LIN {X -288.759,Y -26.804,Z 58.424,A 5.303,B 90.000,C 0.000} C_DIS
LIN {X -288.763,Y -26.761,Z 58.730,A 5.295,B 90.000,C 0.000} C_DIS
LIN {X -288.767,Y -26.710,Z 58.794,A 5.285,B 90.000,C 0.000} C_DIS
LIN {X -288.772,Y -26.660,Z 58.836,A 5.275,B 90.000,C 0.000} C_DIS
LIN {X -288.776,Y -26.617,Z 59.040,A 5.266,B 90.000,C 0.000} C_DIS
LIN {X -288.781,Y -26.567,Z 59.083,A 5.256,B 90.000,C 0.000} C_DIS
LIN {X -288.785,Y -26.516,Z 59.147,A 5.246,B 90.000,C 0.000} C_DIS
LIN {X -288.789,Y -26.473,Z 59.453,A 5.238,B 90.000,C 0.000} C_DIS
LIN {X -288.794,Y -26.423,Z 59.516,A 5.228,B 90.000,C 0.000} C_DIS
LIN {X -288.798,Y -26.372,Z 59.559,A 5.218,B 90.000,C 0.000} C_DIS
LIN {X -288.802,Y -26.330,Z 59.763,A 5.209,B 90.000,C 0.000} C_DIS
LIN {X -288.807,Y -26.279,Z 59.805,A 5.199,B 90.000,C 0.000} C_DIS
LIN {X -288.812,Y -26.228,Z 59.869,A 5.189,B 90.000,C 0.000} C_DIS
LIN {X -288.815,Y -26.186,Z 60.175,A 5.181,B 90.000,C 0.000} C_DIS
LIN {X -288.825,Y -26.084,Z 60.303,A 5.160,B 90.000,C 0.000} C_DIS
LIN {X -288.828,Y -26.042,Z 60.609,A 5.152,B 90.000,C 0.000} C_DIS
LIN {X -288.833,Y -25.991,Z 60.673,A 5.142,B 90.000,C 0.000} C_DIS
LIN {X -288.838,Y -25.940,Z 60.715,A 5.132,B 90.000,C 0.000} C_DIS
LIN {X -288.841,Y -25.898,Z 60.919,A 5.123,B 90.000,C 0.000} C_DIS
LIN {X -288.846,Y -25.847,Z 60.962,A 5.113,B 90.000,C 0.000} C_DIS
LIN {X -288.850,Y -25.796,Z 61.025,A 5.103,B 90.000,C 0.000} C_DIS
LIN {X -288.854,Y -25.754,Z 61.332,A 5.095,B 90.000,C 0.000} C_DIS
LIN {X -288.859,Y -25.703,Z 61.395,A 5.085,B 90.000,C 0.000} C_DIS
LIN {X -288.863,Y -25.652,Z 61.438,A 5.075,B 90.000,C 0.000} C_DIS
LIN {X -288.867,Y -25.610,Z 61.642,A 5.066,B 90.000,C 0.000} C_DIS
LIN {X -288.871,Y -25.559,Z 61.684,A 5.056,B 90.000,C 0.000} C_DIS
LIN {X -288.876,Y -25.508,Z 61.748,A 5.046,B 90.000,C 0.000} C_DIS
LIN {X -288.880,Y -25.466,Z 62.054,A 5.038,B 90.000,C 0.000} C_DIS
LIN {X -288.884,Y -25.415,Z 62.118,A 5.028,B 90.000,C 0.000} C_DIS
LIN {X -288.889,Y -25.364,Z 62.160,A 5.018,B 90.000,C 0.000} C_DIS
LIN {X -288.892,Y -25.322,Z 62.365,A 5.009,B 90.000,C 0.000} C_DIS
LIN {X -288.897,Y -25.271,Z 62.407,A 4.999,B 90.000,C 0.000} C_DIS
LIN {X -288.901,Y -25.220,Z 62.471,A 4.989,B 90.000,C 0.000} C_DIS
LIN {X -288.905,Y -25.178,Z 62.777,A 4.981,B 90.000,C 0.000} C_DIS
LIN {X -288.909,Y -25.127,Z 62.841,A 4.971,B 90.000,C 0.000} C_DIS
LIN {X -288.914,Y -25.076,Z 62.883,A 4.961,B 90.000,C 0.000} C_DIS
LIN {X -288.917,Y -25.034,Z 63.087,A 4.952,B 90.000,C 0.000} C_DIS
LIN {X -288.922,Y -24.983,Z 63.130,A 4.942,B 90.000,C 0.000} C_DIS
LIN {X -288.926,Y -24.932,Z 63.193,A 4.932,B 90.000,C 0.000} C_DIS
LIN {X -288.930,Y -24.890,Z 63.500,A 4.924,B 90.000,C 0.000} C_DIS
LIN {X -288.934,Y -24.839,Z 63.563,A 4.914,B 90.000,C 0.000} C_DIS
LIN {X -288.939,Y -24.788,Z 63.606,A 4.903,B 90.000,C 0.000} C_DIS
LIN {X -288.942,Y -24.746,Z 63.810,A 4.895,B 90.000,C 0.000} C_DIS
LIN {X -288.947,Y -24.695,Z 63.852,A 4.885,B 90.000,C 0.000} C_DIS
LIN {X -288.951,Y -24.644,Z 63.916,A 4.875,B 90.000,C 0.000} C_DIS
LIN {X -288.955,Y -24.602,Z 64.222,A 4.866,B 90.000,C 0.000} C_DIS
LIN {X -288.959,Y -24.551,Z 64.286,A 4.856,B 90.000,C 0.000} C_DIS
LIN {X -288.963,Y -24.500,Z 64.328,A 4.846,B 90.000,C 0.000} C_DIS
LIN {X -288.967,Y -24.458,Z 64.532,A 4.838,B 90.000,C 0.000} C_DIS
LIN {X -288.971,Y -24.407,Z 64.575,A 4.828,B 90.000,C 0.000} C_DIS
LIN {X -288.975,Y -24.356,Z 64.639,A 4.818,B 90.000,C 0.000} C_DIS
LIN {X -288.979,Y -24.314,Z 64.945,A 4.809,B 90.000,C 0.000} C_DIS
LIN {X -288.983,Y -24.263,Z 65.009,A 4.799,B 90.000,C 0.000} C_DIS
LIN {X -288.987,Y -24.212,Z 65.051,A 4.789,B 90.000,C 0.000} C_DIS
LIN {X -288.991,Y -24.170,Z 65.255,A 4.781,B 90.000,C 0.000} C_DIS
LIN {X -288.995,Y -24.119,Z 65.298,A 4.771,B 90.000,C 0.000} C_DIS
LIN {X -289.000,Y -24.068,Z 65.361,A 4.761,B 90.000,C 0.000} C_DIS
LIN {X -289.003,Y -24.026,Z 65.667,A 4.752,B 90.000,C 0.000} C_DIS
LIN {X -289.007,Y -23.975,Z 65.731,A 4.742,B 90.000,C 0.000} C_DIS
LIN {X -289.011,Y -23.924,Z 65.774,A 4.732,B 90.000,C 0.000} C_DIS
LIN {X -289.015,Y -23.882,Z 65.978,A 4.724,B 90.000,C 0.000} C_DIS
LIN {X -289.019,Y -23.831,Z 66.020,A 4.714,B 90.000,C 0.000} C_DIS
LIN {X -289.023,Y -23.780,Z 66.084,A 4.704,B 90.000,C 0.000} C_DIS
LIN {X -289.027,Y -23.738,Z 66.390,A 4.695,B 90.000,C 0.000} C_DIS
LIN {X -289.031,Y -23.687,Z 66.454,A 4.685,B 90.000,C 0.000} C_DIS
LIN {X -289.035,Y -23.636,Z 66.496,A 4.675,B 90.000,C 0.000} C_DIS
LIN {X -289.039,Y -23.594,Z 66.700,A 4.667,B 90.000,C 0.000} C_DIS
LIN {X -289.043,Y -23.543,Z 66.743,A 4.657,B 90.000,C 0.000} C_DIS
LIN {X -289.047,Y -23.492,Z 66.807,A 4.646,B 90.000,C 0.000} C_DIS
LIN {X -289.050,Y -23.450,Z 67.113,A 4.638,B 90.000,C 0.000} C_DIS
LIN {X -289.054,Y -23.399,Z 67.176,A 4.628,B 90.000,C 0.000} C_DIS
LIN {X -289.059,Y -23.348,Z 67.219,A 4.618,B 90.000,C 0.000} C_DIS
LIN {X -289.062,Y -23.306,Z 67.423,A 4.609,B 90.000,C 0.000} C_DIS
LIN {X -289.066,Y -23.255,Z 67.465,A 4.599,B 90.000,C 0.000} C_DIS
LIN {X -289.070,Y -23.204,Z 67.529,A 4.589,B 90.000,C 0.000} C_DIS
LIN {X -289.074,Y -23.162,Z 67.835,A 4.581,B 90.000,C 0.000} C_DIS
LIN {X -289.078,Y -23.111,Z 67.899,A 4.571,B 90.000,C 0.000} C_DIS
LIN {X -289.082,Y -23.060,Z 67.942,A 4.561,B 90.000,C 0.000} C_DIS
LIN {X -289.085,Y -23.017,Z 68.146,A 4.552,B 90.000,C 0.000} C_DIS
LIN {X -289.089,Y -22.967,Z 68.188,A 4.542,B 90.000,C 0.000} C_DIS
LIN {X -289.093,Y -22.916,Z 68.252,A 4.532,B 90.000,C 0.000} C_DIS
LIN {X -289.097,Y -22.873,Z 68.558,A 4.524,B 90.000,C 0.000} C_DIS
LIN {X -289.101,Y -22.822,Z 68.622,A 4.514,B 90.000,C 0.000} C_DIS
LIN {X -289.105,Y -22.772,Z 68.664,A 4.504,B 90.000,C 0.000} C_DIS
LIN {X -289.108,Y -22.729,Z 68.868,A 4.495,B 90.000,C 0.000} C_DIS
LIN {X -289.112,Y -22.678,Z 68.911,A 4.485,B 90.000,C 0.000} C_DIS
LIN {X -289.116,Y -22.628,Z 68.974,A 4.475,B 90.000,C 0.000} C_DIS
LIN {X -289.119,Y -22.585,Z 69.281,A 4.467,B 90.000,C 0.000} C_DIS
LIN {X -289.123,Y -22.534,Z 69.344,A 4.457,B 90.000,C 0.000} C_DIS
LIN {X -289.127,Y -22.483,Z 69.387,A 4.447,B 90.000,C 0.000} C_DIS
LIN {X -289.130,Y -22.441,Z 69.591,A 4.438,B 90.000,C 0.000} C_DIS
LIN {X -289.134,Y -22.390,Z 69.633,A 4.428,B 90.000,C 0.000} C_DIS
LIN {X -289.138,Y -22.339,Z 69.697,A 4.418,B 90.000,C 0.000} C_DIS
LIN {X -289.142,Y -22.297,Z 70.003,A 4.410,B 90.000,C 0.000} C_DIS
LIN {X -289.145,Y -22.246,Z 70.067,A 4.400,B 90.000,C 0.000} C_DIS
LIN {X -289.149,Y -22.195,Z 70.109,A 4.389,B 90.000,C 0.000} C_DIS
LIN {X -289.153,Y -22.153,Z 70.314,A 4.381,B 90.000,C 0.000} C_DIS
LIN {X -289.157,Y -22.102,Z 70.356,A 4.371,B 90.000,C 0.000} C_DIS
LIN {X -289.160,Y -22.051,Z 70.420,A 4.361,B 90.000,C 0.000} C_DIS
LIN {X -289.164,Y -22.009,Z 70.726,A 4.353,B 90.000,C 0.000} C_DIS
LIN {X -289.168,Y -21.958,Z 70.790,A 4.342,B 90.000,C 0.000} C_DIS
LIN {X -289.171,Y -21.907,Z 70.832,A 4.332,B 90.000,C 0.000} C_DIS
LIN {X -289.175,Y -21.865,Z 71.036,A 4.324,B 90.000,C 0.000} C_DIS
LIN {X -289.178,Y -21.814,Z 71.079,A 4.314,B 90.000,C 0.000} C_DIS
LIN {X -289.182,Y -21.763,Z 71.142,A 4.304,B 90.000,C 0.000} C_DIS
LIN {X -289.185,Y -21.721,Z 71.449,A 4.295,B 90.000,C 0.000} C_DIS
LIN {X -289.189,Y -21.670,Z 71.512,A 4.285,B 90.000,C 0.000} C_DIS
LIN {X -289.193,Y -21.619,Z 71.555,A 4.275,B 90.000,C 0.000} C_DIS
LIN {X -289.196,Y -21.576,Z 71.759,A 4.267,B 90.000,C 0.000} C_DIS
LIN {X -289.200,Y -21.526,Z 71.801,A 4.257,B 90.000,C 0.000} C_DIS
LIN {X -289.204,Y -21.475,Z 71.865,A 4.247,B 90.000,C 0.000} C_DIS
LIN {X -289.207,Y -21.432,Z 72.171,A 4.238,B 90.000,C 0.000} C_DIS
LIN {X -289.211,Y -21.381,Z 72.235,A 4.228,B 90.000,C 0.000} C_DIS
LIN {X -289.214,Y -21.331,Z 72.277,A 4.218,B 90.000,C 0.000} C_DIS
LIN {X -289.218,Y -21.288,Z 72.482,A 4.210,B 90.000,C 0.000} C_DIS
LIN {X -289.221,Y -21.237,Z 72.524,A 4.200,B 90.000,C 0.000} C_DIS
LIN {X -289.225,Y -21.186,Z 72.588,A 4.190,B 90.000,C 0.000} C_DIS
LIN {X -289.228,Y -21.144,Z 72.894,A 4.181,B 90.000,C 0.000} C_DIS
LIN {X -289.236,Y -21.042,Z 73.021,A 4.161,B 90.000,C 0.000} C_DIS
LIN {X -289.239,Y -21.000,Z 73.327,A 4.153,B 90.000,C 0.000} C_DIS
LIN {X -289.242,Y -20.949,Z 73.391,A 4.143,B 90.000,C 0.000} C_DIS
LIN {X -289.246,Y -20.898,Z 73.434,A 4.132,B 90.000,C 0.000} C_DIS
LIN {X -289.249,Y -20.856,Z 73.638,A 4.124,B 90.000,C 0.000} C_DIS
LIN {X -289.253,Y -20.805,Z 73.680,A 4.114,B 90.000,C 0.000} C_DIS
LIN {X -289.256,Y -20.754,Z 73.744,A 4.104,B 90.000,C 0.000} C_DIS
LIN {X -289.259,Y -20.712,Z 74.050,A 4.096,B 90.000,C 0.000} C_DIS
LIN {X -289.263,Y -20.661,Z 74.114,A 4.085,B 90.000,C 0.000} C_DIS
LIN {X -289.267,Y -20.610,Z 74.156,A 4.075,B 90.000,C 0.000} C_DIS
LIN {X -289.270,Y -20.567,Z 74.360,A 4.067,B 90.000,C 0.000} C_DIS
LIN {X -289.273,Y -20.517,Z 74.403,A 4.057,B 90.000,C 0.000} C_DIS
LIN {X -289.277,Y -20.466,Z 74.467,A 4.047,B 90.000,C 0.000} C_DIS
LIN {X -289.280,Y -20.423,Z 74.773,A 4.038,B 90.000,C 0.000} C_DIS
LIN {X -289.284,Y -20.372,Z 74.836,A 4.028,B 90.000,C 0.000} C_DIS
LIN {X -289.287,Y -20.321,Z 74.879,A 4.018,B 90.000,C 0.000} C_DIS
LIN {X -289.290,Y -20.279,Z 75.083,A 4.010,B 90.000,C 0.000} C_DIS
LIN {X -289.294,Y -20.228,Z 75.125,A 4.000,B 90.000,C 0.000} C_DIS
LIN {X -289.297,Y -20.177,Z 75.189,A 3.990,B 90.000,C 0.000} C_DIS
LIN {X -289.300,Y -20.135,Z 75.495,A 3.981,B 90.000,C 0.000} C_DIS
LIN {X -289.304,Y -20.084,Z 75.559,A 3.971,B 90.000,C 0.000} C_DIS
LIN {X -289.307,Y -20.033,Z 75.602,A 3.961,B 90.000,C 0.000} C_DIS
LIN {X -289.310,Y -19.991,Z 75.806,A 3.953,B 90.000,C 0.000} C_DIS
LIN {X -289.314,Y -19.940,Z 75.848,A 3.943,B 90.000,C 0.000} C_DIS
LIN {X -289.317,Y -19.889,Z 75.912,A 3.933,B 90.000,C 0.000} C_DIS
LIN {X -289.320,Y -19.847,Z 76.218,A 3.924,B 90.000,C 0.000} C_DIS
LIN {X -289.324,Y -19.796,Z 76.282,A 3.914,B 90.000,C 0.000} C_DIS
LIN {X -289.327,Y -19.745,Z 76.324,A 3.904,B 90.000,C 0.000} C_DIS
LIN {X -289.330,Y -19.702,Z 76.528,A 3.896,B 90.000,C 0.000} C_DIS
LIN {X -289.333,Y -19.651,Z 76.571,A 3.886,B 90.000,C 0.000} C_DIS
LIN {X -289.337,Y -19.601,Z 76.634,A 3.875,B 90.000,C 0.000} C_DIS
LIN {X -289.340,Y -19.558,Z 76.941,A 3.867,B 90.000,C 0.000} C_DIS
LIN {X -289.343,Y -19.507,Z 77.004,A 3.857,B 90.000,C 0.000} C_DIS
LIN {X -289.347,Y -19.456,Z 77.047,A 3.847,B 90.000,C 0.000} C_DIS
LIN {X -289.349,Y -19.414,Z 77.251,A 3.839,B 90.000,C 0.000} C_DIS
LIN {X -289.353,Y -19.363,Z 77.293,A 3.828,B 90.000,C 0.000} C_DIS
LIN {X -289.356,Y -19.312,Z 77.357,A 3.818,B 90.000,C 0.000} C_DIS
LIN {X -289.359,Y -19.270,Z 77.663,A 3.810,B 90.000,C 0.000} C_DIS
LIN {X -289.362,Y -19.219,Z 77.727,A 3.800,B 90.000,C 0.000} C_DIS
LIN {X -289.366,Y -19.168,Z 77.769,A 3.790,B 90.000,C 0.000} C_DIS
LIN {X -289.369,Y -19.126,Z 77.974,A 3.781,B 90.000,C 0.000} C_DIS
LIN {X -289.372,Y -19.075,Z 78.016,A 3.771,B 90.000,C 0.000} C_DIS
LIN {X -289.375,Y -19.024,Z 78.080,A 3.761,B 90.000,C 0.000} C_DIS
LIN {X -289.378,Y -18.981,Z 78.386,A 3.753,B 90.000,C 0.000} C_DIS
LIN {X -289.381,Y -18.930,Z 78.450,A 3.743,B 90.000,C 0.000} C_DIS
LIN {X -289.385,Y -18.879,Z 78.492,A 3.733,B 90.000,C 0.000} C_DIS
LIN {X -289.388,Y -18.837,Z 78.696,A 3.724,B 90.000,C 0.000} C_DIS
LIN {X -289.391,Y -18.786,Z 78.739,A 3.714,B 90.000,C 0.000} C_DIS
LIN {X -289.394,Y -18.735,Z 78.802,A 3.704,B 90.000,C 0.000} C_DIS
LIN {X -289.397,Y -18.693,Z 79.109,A 3.696,B 90.000,C 0.000} C_DIS
LIN {X -289.400,Y -18.642,Z 79.172,A 3.686,B 90.000,C 0.000} C_DIS
LIN {X -289.403,Y -18.591,Z 79.215,A 3.676,B 90.000,C 0.000} C_DIS
LIN {X -289.406,Y -18.549,Z 79.419,A 3.667,B 90.000,C 0.000} C_DIS
LIN {X -289.409,Y -18.498,Z 79.461,A 3.657,B 90.000,C 0.000} C_DIS
LIN {X -289.413,Y -18.447,Z 79.525,A 3.647,B 90.000,C 0.000} C_DIS
LIN {X -289.415,Y -18.404,Z 79.831,A 3.639,B 90.000,C 0.000} C_DIS
LIN {X -289.419,Y -18.353,Z 79.895,A 3.629,B 90.000,C 0.000} C_DIS
LIN {X -289.422,Y -18.303,Z 79.937,A 3.618,B 90.000,C 0.000} C_DIS
LIN {X -289.425,Y -18.260,Z 80.142,A 3.610,B 90.000,C 0.000} C_DIS
LIN {X -289.428,Y -18.209,Z 80.184,A 3.600,B 90.000,C 0.000} C_DIS
LIN {X -289.431,Y -18.158,Z 80.248,A 3.590,B 90.000,C 0.000} C_DIS
LIN {X -289.434,Y -18.116,Z 80.554,A 3.582,B 90.000,C 0.000} C_DIS
LIN {X -289.437,Y -18.065,Z 80.618,A 3.571,B 90.000,C 0.000} C_DIS
LIN {X -289.440,Y -18.014,Z 80.660,A 3.561,B 90.000,C 0.000} C_DIS
LIN {X -289.443,Y -17.972,Z 80.864,A 3.553,B 90.000,C 0.000} C_DIS
LIN {X -289.446,Y -17.921,Z 80.907,A 3.543,B 90.000,C 0.000} C_DIS
LIN {X -289.449,Y -17.870,Z 80.970,A 3.533,B 90.000,C 0.000} C_DIS
LIN {X -289.452,Y -17.827,Z 81.277,A 3.524,B 90.000,C 0.000} C_DIS
LIN {X -289.455,Y -17.776,Z 81.340,A 3.514,B 90.000,C 0.000} C_DIS
LIN {X -289.458,Y -17.726,Z 81.383,A 3.504,B 90.000,C 0.000} C_DIS
LIN {X -289.460,Y -17.683,Z 81.587,A 3.496,B 90.000,C 0.000} C_DIS
LIN {X -289.463,Y -17.632,Z 81.629,A 3.486,B 90.000,C 0.000} C_DIS
LIN {X -289.467,Y -17.581,Z 81.693,A 3.476,B 90.000,C 0.000} C_DIS
LIN {X -289.469,Y -17.539,Z 81.999,A 3.467,B 90.000,C 0.000} C_DIS
LIN {X -289.472,Y -17.488,Z 82.063,A 3.457,B 90.000,C 0.000} C_DIS
LIN {X -289.475,Y -17.437,Z 82.105,A 3.447,B 90.000,C 0.000} C_DIS
LIN {X -289.478,Y -17.395,Z 82.309,A 3.439,B 90.000,C 0.000} C_DIS
LIN {X -289.481,Y -17.344,Z 82.352,A 3.429,B 90.000,C 0.000} C_DIS
LIN {X -289.484,Y -17.293,Z 82.416,A 3.419,B 90.000,C 0.000} C_DIS
LIN {X -289.486,Y -17.250,Z 82.722,A 3.410,B 90.000,C 0.000} C_DIS
LIN {X -289.490,Y -17.199,Z 82.785,A 3.400,B 90.000,C 0.000} C_DIS
LIN {X -289.493,Y -17.148,Z 82.828,A 3.390,B 90.000,C 0.000} C_DIS
LIN {X -289.495,Y -17.106,Z 83.032,A 3.382,B 90.000,C 0.000} C_DIS
LIN {X -289.498,Y -17.055,Z 83.075,A 3.372,B 90.000,C 0.000} C_DIS
LIN {X -289.501,Y -17.004,Z 83.138,A 3.361,B 90.000,C 0.000} C_DIS
LIN {X -289.504,Y -16.962,Z 83.444,A 3.353,B 90.000,C 0.000} C_DIS
LIN {X -289.507,Y -16.911,Z 83.508,A 3.343,B 90.000,C 0.000} C_DIS
LIN {X -289.509,Y -16.860,Z 83.551,A 3.333,B 90.000,C 0.000} C_DIS
LIN {X -289.512,Y -16.818,Z 83.755,A 3.325,B 90.000,C 0.000} C_DIS
LIN {X -289.515,Y -16.767,Z 83.797,A 3.314,B 90.000,C 0.000} C_DIS
LIN {X -289.518,Y -16.716,Z 83.861,A 3.304,B 90.000,C 0.000} C_DIS
LIN {X -289.520,Y -16.673,Z 84.167,A 3.296,B 90.000,C 0.000} C_DIS
LIN {X -289.523,Y -16.622,Z 84.231,A 3.286,B 90.000,C 0.000} C_DIS
LIN {X -289.526,Y -16.571,Z 84.273,A 3.276,B 90.000,C 0.000} C_DIS
LIN {X -289.529,Y -16.529,Z 84.477,A 3.267,B 90.000,C 0.000} C_DIS
LIN {X -289.531,Y -16.478,Z 84.520,A 3.257,B 90.000,C 0.000} C_DIS
LIN {X -289.534,Y -16.427,Z 84.584,A 3.247,B 90.000,C 0.000} C_DIS
LIN {X -289.537,Y -16.385,Z 84.890,A 3.239,B 90.000,C 0.000} C_DIS
LIN {X -289.543,Y -16.283,Z 85.017,A 3.219,B 90.000,C 0.000} C_DIS
LIN {X -289.545,Y -16.240,Z 85.323,A 3.210,B 90.000,C 0.000} C_DIS
LIN {X -289.548,Y -16.189,Z 85.387,A 3.200,B 90.000,C 0.000} C_DIS
LIN {X -289.551,Y -16.138,Z 85.429,A 3.190,B 90.000,C 0.000} C_DIS
LIN {X -289.553,Y -16.096,Z 85.634,A 3.182,B 90.000,C 0.000} C_DIS
LIN {X -289.556,Y -16.045,Z 85.676,A 3.172,B 90.000,C 0.000} C_DIS
LIN {X -289.559,Y -15.994,Z 85.740,A 3.162,B 90.000,C 0.000} C_DIS
LIN {X -289.561,Y -15.952,Z 86.046,A 3.153,B 90.000,C 0.000} C_DIS
LIN {X -289.564,Y -15.901,Z 86.110,A 3.143,B 90.000,C 0.000} C_DIS
LIN {X -289.567,Y -15.850,Z 86.152,A 3.133,B 90.000,C 0.000} C_DIS
LIN {X -289.569,Y -15.807,Z 86.356,A 3.125,B 90.000,C 0.000} C_DIS
LIN {X -289.572,Y -15.756,Z 86.399,A 3.115,B 90.000,C 0.000} C_DIS
LIN {X -289.574,Y -15.706,Z 86.462,A 3.104,B 90.000,C 0.000} C_DIS
LIN {X -289.577,Y -15.663,Z 86.769,A 3.096,B 90.000,C 0.000} C_DIS
LIN {X -289.579,Y -15.612,Z 86.832,A 3.086,B 90.000,C 0.000} C_DIS
LIN {X -289.582,Y -15.561,Z 86.875,A 3.076,B 90.000,C 0.000} C_DIS
LIN {X -289.584,Y -15.519,Z 87.079,A 3.068,B 90.000,C 0.000} C_DIS
LIN {X -289.587,Y -15.468,Z 87.121,A 3.057,B 90.000,C 0.000} C_DIS
LIN {X -289.590,Y -15.417,Z 87.185,A 3.047,B 90.000,C 0.000} C_DIS
LIN {X -289.592,Y -15.374,Z 87.491,A 3.039,B 90.000,C 0.000} C_DIS
LIN {X -289.595,Y -15.324,Z 87.555,A 3.029,B 90.000,C 0.000} C_DIS
LIN {X -289.598,Y -15.273,Z 87.597,A 3.019,B 90.000,C 0.000} C_DIS
LIN {X -289.600,Y -15.230,Z 87.802,A 3.010,B 90.000,C 0.000} C_DIS
LIN {X -289.602,Y -15.179,Z 87.844,A 3.000,B 90.000,C 0.000} C_DIS
LIN {X -289.605,Y -15.128,Z 87.908,A 2.990,B 90.000,C 0.000} C_DIS
LIN {X -289.607,Y -15.086,Z 88.214,A 2.982,B 90.000,C 0.000} C_DIS
LIN {X -289.610,Y -15.035,Z 88.278,A 2.972,B 90.000,C 0.000} C_DIS
LIN {X -289.613,Y -14.984,Z 88.320,A 2.962,B 90.000,C 0.000} C_DIS
LIN {X -289.615,Y -14.941,Z 88.524,A 2.953,B 90.000,C 0.000} C_DIS
LIN {X -289.617,Y -14.891,Z 88.567,A 2.943,B 90.000,C 0.000} C_DIS
LIN {X -289.620,Y -14.840,Z 88.630,A 2.933,B 90.000,C 0.000} C_DIS
LIN {X -289.622,Y -14.797,Z 88.937,A 2.925,B 90.000,C 0.000} C_DIS
LIN {X -289.625,Y -14.746,Z 89.000,A 2.915,B 90.000,C 0.000} C_DIS
LIN {X -289.627,Y -14.695,Z 89.043,A 2.905,B 90.000,C 0.000} C_DIS
LIN {X -289.630,Y -14.653,Z 89.247,A 2.896,B 90.000,C 0.000} C_DIS
LIN {X -289.632,Y -14.602,Z 89.289,A 2.886,B 90.000,C 0.000} C_DIS
LIN {X -289.635,Y -14.551,Z 89.353,A 2.876,B 90.000,C 0.000} C_DIS
LIN {X -289.637,Y -14.508,Z 89.659,A 2.868,B 90.000,C 0.000} C_DIS
LIN {X -289.639,Y -14.457,Z 89.723,A 2.858,B 90.000,C 0.000} C_DIS
LIN {X -289.642,Y -14.407,Z 89.765,A 2.847,B 90.000,C 0.000} C_DIS
LIN {X -289.644,Y -14.364,Z 89.969,A 2.839,B 90.000,C 0.000} C_DIS
LIN {X -289.647,Y -14.313,Z 90.012,A 2.829,B 90.000,C 0.000} C_DIS
LIN {X -289.649,Y -14.262,Z 90.076,A 2.819,B 90.000,C 0.000} C_DIS
LIN {X -289.651,Y -14.220,Z 90.382,A 2.811,B 90.000,C 0.000} C_DIS
LIN {X -289.654,Y -14.169,Z 90.445,A 2.800,B 90.000,C 0.000} C_DIS
LIN {X -289.656,Y -14.118,Z 90.488,A 2.790,B 90.000,C 0.000} C_DIS
LIN {X -289.658,Y -14.075,Z 90.692,A 2.782,B 90.000,C 0.000} C_DIS
LIN {X -289.661,Y -14.024,Z 90.735,A 2.772,B 90.000,C 0.000} C_DIS
LIN {X -289.663,Y -13.973,Z 90.798,A 2.762,B 90.000,C 0.000} C_DIS
LIN {X -289.665,Y -13.931,Z 91.104,A 2.753,B 90.000,C 0.000} C_DIS
LIN {X -289.668,Y -13.880,Z 91.168,A 2.743,B 90.000,C 0.000} C_DIS
LIN {X -289.670,Y -13.829,Z 91.211,A 2.733,B 90.000,C 0.000} C_DIS
LIN {X -289.672,Y -13.787,Z 91.415,A 2.725,B 90.000,C 0.000} C_DIS
LIN {X -289.675,Y -13.736,Z 91.457,A 2.715,B 90.000,C 0.000} C_DIS
LIN {X -289.677,Y -13.685,Z 91.521,A 2.705,B 90.000,C 0.000} C_DIS
LIN {X -289.679,Y -13.642,Z 91.827,A 2.696,B 90.000,C 0.000} C_DIS
LIN {X -289.681,Y -13.591,Z 91.891,A 2.686,B 90.000,C 0.000} C_DIS
LIN {X -289.684,Y -13.540,Z 91.933,A 2.676,B 90.000,C 0.000} C_DIS
LIN {X -289.686,Y -13.498,Z 92.137,A 2.668,B 90.000,C 0.000} C_DIS
LIN {X -289.688,Y -13.447,Z 92.180,A 2.658,B 90.000,C 0.000} C_DIS
LIN {X -289.690,Y -13.396,Z 92.244,A 2.648,B 90.000,C 0.000} C_DIS
LIN {X -289.692,Y -13.354,Z 92.550,A 2.639,B 90.000,C 0.000} C_DIS
LIN {X -289.695,Y -13.303,Z 92.613,A 2.629,B 90.000,C 0.000} C_DIS
LIN {X -289.697,Y -13.252,Z 92.656,A 2.619,B 90.000,C 0.000} C_DIS
LIN {X -289.699,Y -13.209,Z 92.860,A 2.611,B 90.000,C 0.000} C_DIS
LIN {X -289.701,Y -13.158,Z 92.902,A 2.601,B 90.000,C 0.000} C_DIS
LIN {X -289.704,Y -13.107,Z 92.966,A 2.590,B 90.000,C 0.000} C_DIS
LIN {X -289.706,Y -13.065,Z 93.272,A 2.582,B 90.000,C 0.000} C_DIS
LIN {X -289.708,Y -13.014,Z 93.336,A 2.572,B 90.000,C 0.000} C_DIS
LIN {X -289.710,Y -12.963,Z 93.379,A 2.562,B 90.000,C 0.000} C_DIS
LIN {X -289.712,Y -12.920,Z 93.583,A 2.554,B 90.000,C 0.000} C_DIS
LIN {X -289.714,Y -12.869,Z 93.625,A 2.543,B 90.000,C 0.000} C_DIS
LIN {X -289.717,Y -12.818,Z 93.689,A 2.533,B 90.000,C 0.000} C_DIS
LIN {X -289.718,Y -12.776,Z 93.995,A 2.525,B 90.000,C 0.000} C_DIS
LIN {X -289.721,Y -12.725,Z 94.059,A 2.515,B 90.000,C 0.000} C_DIS
LIN {X -289.723,Y -12.674,Z 94.101,A 2.505,B 90.000,C 0.000} C_DIS
LIN {X -289.725,Y -12.632,Z 94.305,A 2.496,B 90.000,C 0.000} C_DIS
LIN {X -289.727,Y -12.581,Z 94.348,A 2.486,B 90.000,C 0.000} C_DIS
LIN {X -289.729,Y -12.530,Z 94.411,A 2.476,B 90.000,C 0.000} C_DIS
LIN {X -289.731,Y -12.487,Z 94.718,A 2.468,B 90.000,C 0.000} C_DIS
LIN {X -289.733,Y -12.436,Z 94.781,A 2.458,B 90.000,C 0.000} C_DIS
LIN {X -289.735,Y -12.385,Z 94.824,A 2.448,B 90.000,C 0.000} C_DIS
LIN {X -289.737,Y -12.343,Z 95.028,A 2.439,B 90.000,C 0.000} C_DIS
LIN {X -289.739,Y -12.292,Z 95.070,A 2.429,B 90.000,C 0.000} C_DIS
LIN {X -289.742,Y -12.241,Z 95.134,A 2.419,B 90.000,C 0.000} C_DIS
LIN {X -289.743,Y -12.198,Z 95.440,A 2.411,B 90.000,C 0.000} C_DIS
LIN {X -289.745,Y -12.147,Z 95.504,A 2.401,B 90.000,C 0.000} C_DIS
LIN {X -289.748,Y -12.096,Z 95.546,A 2.391,B 90.000,C 0.000} C_DIS
LIN {X -289.749,Y -12.054,Z 95.751,A 2.382,B 90.000,C 0.000} C_DIS
LIN {X -289.751,Y -12.003,Z 95.793,A 2.372,B 90.000,C 0.000} C_DIS
LIN {X -289.754,Y -11.952,Z 95.857,A 2.362,B 90.000,C 0.000} C_DIS
LIN {X -289.755,Y -11.910,Z 96.163,A 2.354,B 90.000,C 0.000} C_DIS
LIN {X -289.757,Y -11.859,Z 96.227,A 2.344,B 90.000,C 0.000} C_DIS
LIN {X -289.760,Y -11.808,Z 96.269,A 2.334,B 90.000,C 0.000} C_DIS
LIN {X -289.761,Y -11.765,Z 96.473,A 2.325,B 90.000,C 0.000} C_DIS
LIN {X -289.763,Y -11.714,Z 96.516,A 2.315,B 90.000,C 0.000} C_DIS
LIN {X -289.765,Y -11.663,Z 96.579,A 2.305,B 90.000,C 0.000} C_DIS
LIN {X -289.767,Y -11.621,Z 96.886,A 2.297,B 90.000,C 0.000} C_DIS
LIN {X -289.769,Y -11.570,Z 96.949,A 2.286,B 90.000,C 0.000} C_DIS
LIN {X -289.771,Y -11.519,Z 96.992,A 2.276,B 90.000,C 0.000} C_DIS
LIN {X -289.773,Y -11.476,Z 97.196,A 2.268,B 90.000,C 0.000} C_DIS
LIN {X -289.775,Y -11.425,Z 97.238,A 2.258,B 90.000,C 0.000} C_DIS
LIN {X -289.777,Y -11.374,Z 97.302,A 2.248,B 90.000,C 0.000} C_DIS
LIN {X -289.779,Y -11.332,Z 97.608,A 2.239,B 90.000,C 0.000} C_DIS
LIN {X -289.782,Y -11.230,Z 97.736,A 2.219,B 90.000,C 0.000} C_DIS
LIN {X -289.784,Y -11.188,Z 98.042,A 2.211,B 90.000,C 0.000} C_DIS
LIN {X -289.786,Y -11.137,Z 98.105,A 2.201,B 90.000,C 0.000} C_DIS
LIN {X -289.788,Y -11.086,Z 98.148,A 2.191,B 90.000,C 0.000} C_DIS
LIN {X -289.790,Y -11.043,Z 98.352,A 2.182,B 90.000,C 0.000} C_DIS
LIN {X -289.792,Y -10.992,Z 98.395,A 2.172,B 90.000,C 0.000} C_DIS
LIN {X -289.794,Y -10.941,Z 98.458,A 2.162,B 90.000,C 0.000} C_DIS
LIN {X -289.795,Y -10.899,Z 98.764,A 2.154,B 90.000,C 0.000} C_DIS
LIN {X -289.797,Y -10.848,Z 98.828,A 2.144,B 90.000,C 0.000} C_DIS
LIN {X -289.799,Y -10.797,Z 98.871,A 2.134,B 90.000,C 0.000} C_DIS
LIN {X -289.801,Y -10.754,Z 99.075,A 2.125,B 90.000,C 0.000} C_DIS
LIN {X -289.802,Y -10.703,Z 99.117,A 2.115,B 90.000,C 0.000} C_DIS
LIN {X -289.804,Y -10.652,Z 99.181,A 2.105,B 90.000,C 0.000} C_DIS
LIN {X -289.806,Y -10.610,Z 99.487,A 2.097,B 90.000,C 0.000} C_DIS
LIN {X -289.808,Y -10.559,Z 99.551,A 2.087,B 90.000,C 0.000} C_DIS
LIN {X -289.810,Y -10.508,Z 99.593,A 2.077,B 90.000,C 0.000} C_DIS
LIN {X -289.811,Y -10.465,Z 99.797,A 2.068,B 90.000,C 0.000} C_DIS
LIN {X -289.813,Y -10.414,Z 99.840,A 2.058,B 90.000,C 0.000} C_DIS
LIN {X -289.815,Y -10.363,Z 99.904,A 2.048,B 90.000,C 0.000} C_DIS
LIN {X -289.816,Y -10.321,Z 100.210,A 2.040,B 90.000,C 0.000} C_DIS
LIN {X -289.818,Y -10.270,Z 100.273,A 2.029,B 90.000,C 0.000} C_DIS
LIN {X -289.820,Y -10.219,Z 100.316,A 2.019,B 90.000,C 0.000} C_DIS
LIN {X -289.821,Y -10.177,Z 100.520,A 2.011,B 90.000,C 0.000} C_DIS
LIN {X -289.823,Y -10.126,Z 100.562,A 2.001,B 90.000,C 0.000} C_DIS
LIN {X -289.825,Y -10.075,Z 100.626,A 1.991,B 90.000,C 0.000} C_DIS
LIN {X -289.826,Y -10.032,Z 100.932,A 1.982,B 90.000,C 0.000} C_DIS
LIN {X -289.828,Y -9.981,Z 100.996,A 1.972,B 90.000,C 0.000} C_DIS
LIN {X -289.830,Y -9.930,Z 101.039,A 1.962,B 90.000,C 0.000} C_DIS
LIN {X -289.831,Y -9.888,Z 101.243,A 1.954,B 90.000,C 0.000} C_DIS
LIN {X -289.833,Y -9.837,Z 101.285,A 1.944,B 90.000,C 0.000} C_DIS
LIN {X -289.835,Y -9.786,Z 101.349,A 1.934,B 90.000,C 0.000} C_DIS
LIN {X -289.836,Y -9.743,Z 101.655,A 1.925,B 90.000,C 0.000} C_DIS
LIN {X -289.838,Y -9.692,Z 101.719,A 1.915,B 90.000,C 0.000} C_DIS
LIN {X -289.840,Y -9.641,Z 101.761,A 1.905,B 90.000,C 0.000} C_DIS
LIN {X -289.841,Y -9.599,Z 101.965,A 1.897,B 90.000,C 0.000} C_DIS
LIN {X -289.843,Y -9.548,Z 102.008,A 1.887,B 90.000,C 0.000} C_DIS
LIN {X -289.844,Y -9.497,Z 102.071,A 1.877,B 90.000,C 0.000} C_DIS
LIN {X -289.846,Y -9.454,Z 102.378,A 1.868,B 90.000,C 0.000} C_DIS
LIN {X -289.848,Y -9.403,Z 102.441,A 1.858,B 90.000,C 0.000} C_DIS
LIN {X -289.849,Y -9.352,Z 102.484,A 1.848,B 90.000,C 0.000} C_DIS
LIN {X -289.851,Y -9.310,Z 102.688,A 1.840,B 90.000,C 0.000} C_DIS
LIN {X -289.852,Y -9.259,Z 102.730,A 1.830,B 90.000,C 0.000} C_DIS
LIN {X -289.854,Y -9.208,Z 102.794,A 1.820,B 90.000,C 0.000} C_DIS
LIN {X -289.855,Y -9.165,Z 103.100,A 1.811,B 90.000,C 0.000} C_DIS
LIN {X -289.857,Y -9.114,Z 103.164,A 1.801,B 90.000,C 0.000} C_DIS
LIN {X -289.858,Y -9.063,Z 103.206,A 1.791,B 90.000,C 0.000} C_DIS
LIN {X -289.860,Y -9.021,Z 103.411,A 1.783,B 90.000,C 0.000} C_DIS
LIN {X -289.861,Y -8.970,Z 103.453,A 1.772,B 90.000,C 0.000} C_DIS
LIN {X -289.863,Y -8.919,Z 103.517,A 1.762,B 90.000,C 0.000} C_DIS
LIN {X -289.864,Y -8.877,Z 103.823,A 1.754,B 90.000,C 0.000} C_DIS
LIN {X -289.866,Y -8.826,Z 103.887,A 1.744,B 90.000,C 0.000} C_DIS
LIN {X -289.867,Y -8.775,Z 103.929,A 1.734,B 90.000,C 0.000} C_DIS
LIN {X -289.869,Y -8.732,Z 104.133,A 1.725,B 90.000,C 0.000} C_DIS
LIN {X -289.870,Y -8.681,Z 104.176,A 1.715,B 90.000,C 0.000} C_DIS
LIN {X -289.872,Y -8.630,Z 104.238,A 1.705,B 90.000,C 0.000} C_DIS
LIN {X -289.873,Y -8.582,Z 104.545,A 1.696,B 90.000,C 0.000} C_DIS
LIN {X -289.875,Y -8.519,Z 104.629,A 1.683,B 90.000,C 0.000} C_DIS
LIN {X -289.876,Y -8.470,Z 104.668,A 1.674,B 90.000,C 0.000} C_DIS
RET=EKI_SetBool("oxy","torchState",FALSE)
RET = EKI_Send("oxy","torchState")
PTP {X -287.877,Y -8.411,Z 104.668,A 1.674,B 90.000,C 0.000}
PTP {X -269.885,Y -7.886,Z 104.668,A 1.674,B 90.000,C 0.000}
PTP {X -264.196,Y 55.683,Z 65.409,A -11.902,B 90.000,C 0.000}
PTP {X -281.809,Y 59.395,Z 65.409,A -11.902,B 90.000,C 0.000}
WAIT SEC 2
RET=EKI_SetBool("oxy","torchState",TRUE)
RET = EKI_Send("oxy","torchState")
LIN {X -283.766,Y 59.808,Z 65.409,A -11.902,B 90.000,C 0.000} C_DIS
LIN {X -283.766,Y 59.808,Z 65.409,A -11.902,B 90.000,C 0.000} C_DIS
RET=EKI_SetBool("oxy","torchState",FALSE)
RET = EKI_Send("oxy","torchState")
PTP {X -281.809,Y 59.395,Z 65.409,A -11.902,B 90.000,C 0.000}
PTP {X -264.196,Y 55.683,Z 65.409,A -11.902,B 90.000,C 0.000}
PTP {X -205.108,Y -175.587,Z 134.156,A 40.566,B 90.000,C 0.000}
PTP {X -218.782,Y -187.293,Z 134.156,A 40.566,B 90.000,C 0.000}
WAIT SEC 2
RET=EKI_SetBool("oxy","torchState",TRUE)
RET = EKI_Send("oxy","torchState")
LIN {X -220.301,Y -188.593,Z 134.156,A 40.566,B 90.000,C 0.000} C_DIS
LIN {X -220.295,Y -188.601,Z 133.387,A 40.568,B 90.000,C 0.000} C_DIS
LIN {X -220.203,Y -188.708,Z 132.591,A 40.596,B 90.000,C 0.000} C_DIS
LIN {X -219.627,Y -189.377,Z 130.252,A 40.770,B 90.000,C 0.000} C_DIS
LIN {X -219.299,Y -189.758,Z 128.994,A 40.869,B 90.000,C 0.000} C_DIS
LIN {X -218.964,Y -190.144,Z 126.547,A 40.970,B 90.000,C 0.000} C_DIS
LIN {X -218.825,Y -190.304,Z 124.056,A 41.012,B 90.000,C 0.000} C_DIS
LIN {X -218.737,Y -190.406,Z 121.560,A 41.039,B 90.000,C 0.000} C_DIS
LIN {X -218.677,Y -190.474,Z 120.080,A 41.057,B 90.000,C 0.000} C_DIS
LIN {X -218.307,Y -190.898,Z 117.645,A 41.168,B 90.000,C 0.000} C_DIS
LIN {X -218.004,Y -191.244,Z 116.378,A 41.259,B 90.000,C 0.000} C_DIS
LIN {X -217.687,Y -191.605,Z 115.423,A 41.354,B 90.000,C 0.000} C_DIS
LIN {X -217.268,Y -192.080,Z 114.509,A 41.479,B 90.000,C 0.000} C_DIS
LIN {X -216.771,Y -192.640,Z 113.712,A 41.627,B 90.000,C 0.000} C_DIS
LIN {X -216.193,Y -193.289,Z 113.030,A 41.799,B 90.000,C 0.000} C_DIS
LIN {X -215.532,Y -194.026,Z 112.461,A 41.994,B 90.000,C 0.000} C_DIS
LIN {X -214.746,Y -194.895,Z 111.969,A 42.226,B 90.000,C 0.000} C_DIS
LIN {X -213.126,Y -196.664,Z 111.264,A 42.700,B 90.000,C 0.000} C_DIS
LIN {X -212.795,Y -197.023,Z 111.119,A 42.796,B 90.000,C 0.000} C_DIS
LIN {X -212.233,Y -197.629,Z 110.702,A 42.959,B 90.000,C 0.000} C_DIS
LIN {X -211.874,Y -198.014,Z 110.108,A 43.063,B 90.000,C 0.000} C_DIS
LIN {X -211.579,Y -198.329,Z 109.184,A 43.149,B 90.000,C 0.000} C_DIS
LIN {X -211.136,Y -198.800,Z 106.769,A 43.276,B 90.000,C 0.000} C_DIS
LIN {X -210.874,Y -199.078,Z 104.298,A 43.352,B 90.000,C 0.000} C_DIS
LIN {X -210.622,Y -199.345,Z 101.825,A 43.424,B 90.000,C 0.000} C_DIS
LIN {X -210.348,Y -199.633,Z 99.357,A 43.503,B 90.000,C 0.000} C_DIS
LIN {X -210.033,Y -199.965,Z 96.900,A 43.593,B 90.000,C 0.000} C_DIS
LIN {X -209.700,Y -200.315,Z 94.447,A 43.689,B 90.000,C 0.000} C_DIS
LIN {X -209.345,Y -200.685,Z 92.000,A 43.790,B 90.000,C 0.000} C_DIS
LIN {X -209.008,Y -201.037,Z 89.877,A 43.886,B 90.000,C 0.000} C_DIS
LIN {X -208.478,Y -201.586,Z 87.799,A 44.037,B 90.000,C 0.000} C_DIS
LIN {X -207.598,Y -202.491,Z 85.641,A 44.287,B 90.000,C 0.000} C_DIS
LIN {X -206.553,Y -203.550,Z 83.632,A 44.580,B 90.000,C 0.000} C_DIS
LIN {X -205.476,Y -204.635,Z 81.654,A 44.882,B 90.000,C 0.000} C_DIS
LIN {X -204.399,Y -205.720,Z 79.676,A 45.185,B 90.000,C 0.000} C_DIS
LIN {X -203.301,Y -206.801,Z 77.707,A 45.489,B 90.000,C 0.000} C_DIS
LIN {X -202.204,Y -207.878,Z 75.737,A 45.793,B 90.000,C 0.000} C_DIS
LIN {X -201.136,Y -208.910,Z 73.725,A 46.086,B 90.000,C 0.000} C_DIS
LIN {X -200.113,Y -209.890,Z 71.666,A 46.366,B 90.000,C 0.000} C_DIS
LIN {X -199.145,Y -210.810,Z 69.552,A 46.630,B 90.000,C 0.000} C_DIS
LIN {X -198.215,Y -211.685,Z 67.403,A 46.882,B 90.000,C 0.000} C_DIS
LIN {X -197.292,Y -212.546,Z 65.245,A 47.131,B 90.000,C 0.000} C_DIS
LIN {X -196.393,Y -213.377,Z 63.065,A 47.373,B 90.000,C 0.000} C_DIS
LIN {X -195.630,Y -214.077,Z 61.129,A 47.578,B 90.000,C 0.000} C_DIS
LIN {X -194.473,Y -215.128,Z 59.401,A 47.887,B 90.000,C 0.000} C_DIS
LIN {X -193.006,Y -216.445,Z 57.863,A 48.276,B 90.000,C 0.000} C_DIS
LIN {X -192.258,Y -217.110,Z 57.133,A 48.474,B 90.000,C 0.000} C_DIS
LIN {X -191.704,Y -217.599,Z 56.704,A 48.620,B 90.000,C 0.000} C_DIS
LIN {X -191.032,Y -218.190,Z 56.365,A 48.797,B 90.000,C 0.000} C_DIS
LIN {X -190.345,Y -218.790,Z 56.183,A 48.977,B 90.000,C 0.000} C_DIS
LIN {X -189.810,Y -219.254,Z 56.184,A 49.117,B 90.000,C 0.000} C_DIS
LIN {X -189.652,Y -219.390,Z 56.261,A 49.158,B 90.000,C 0.000} C_DIS
LIN {X -189.595,Y -219.440,Z 56.392,A 49.173,B 90.000,C 0.000} C_DIS
LIN {X -189.727,Y -219.325,Z 56.810,A 49.139,B 90.000,C 0.000} C_DIS
LIN {X -190.641,Y -218.532,Z 58.246,A 48.899,B 90.000,C 0.000} C_DIS
LIN {X -190.847,Y -218.352,Z 59.007,A 48.845,B 90.000,C 0.000} C_DIS
LIN {X -190.927,Y -218.281,Z 59.857,A 48.824,B 90.000,C 0.000} C_DIS
LIN {X -190.881,Y -218.322,Z 60.761,A 48.837,B 90.000,C 0.000} C_DIS
LIN {X -190.707,Y -218.474,Z 61.684,A 48.882,B 90.000,C 0.000} C_DIS
LIN {X -190.384,Y -218.755,Z 62.648,A 48.967,B 90.000,C 0.000} C_DIS
LIN {X -189.914,Y -219.164,Z 63.572,A 49.090,B 90.000,C 0.000} C_DIS
LIN {X -189.271,Y -219.719,Z 64.495,A 49.258,B 90.000,C 0.000} C_DIS
LIN {X -187.877,Y -220.912,Z 66.084,A 49.620,B 90.000,C 0.000} C_DIS
LIN {X -187.473,Y -221.255,Z 66.655,A 49.725,B 90.000,C 0.000} C_DIS
LIN {X -187.195,Y -221.490,Z 67.210,A 49.797,B 90.000,C 0.000} C_DIS
LIN {X -187.019,Y -221.639,Z 67.789,A 49.842,B 90.000,C 0.000} C_DIS
LIN {X -186.969,Y -221.681,Z 68.415,A 49.855,B 90.000,C 0.000} C_DIS
LIN {X -187.101,Y -221.570,Z 69.043,A 49.821,B 90.000,C 0.000} C_DIS
LIN {X -187.434,Y -221.288,Z 69.695,A 49.735,B 90.000,C 0.000} C_DIS
LIN {X -188.841,Y -220.088,Z 71.377,A 49.370,B 90.000,C 0.000} C_DIS
LIN {X -189.138,Y -219.833,Z 71.740,A 49.292,B 90.000,C 0.000} C_DIS
LIN {X -189.376,Y -219.629,Z 72.332,A 49.230,B 90.000,C 0.000} C_DIS
LIN {X -189.576,Y -219.456,Z 73.148,A 49.178,B 90.000,C 0.000} C_DIS
LIN {X -189.794,Y -219.267,Z 75.632,A 49.121,B 90.000,C 0.000} C_DIS
LIN {X -189.793,Y -219.269,Z 76.089,A 49.121,B 90.000,C 0.000} C_DIS
LIN {X -189.711,Y -219.339,Z 76.355,A 49.143,B 90.000,C 0.000} C_DIS
LIN {X -189.592,Y -219.443,Z 76.470,A 49.174,B 90.000,C 0.000} C_DIS
LIN {X -189.434,Y -219.579,Z 76.283,A 49.215,B 90.000,C 0.000} C_DIS
LIN {X -189.047,Y -219.912,Z 74.946,A 49.316,B 90.000,C 0.000} C_DIS
LIN {X -188.750,Y -220.167,Z 74.169,A 49.393,B 90.000,C 0.000} C_DIS
LIN {X -187.877,Y -220.912,Z 72.569,A 49.620,B 90.000,C 0.000} C_DIS
LIN {X -187.015,Y -221.642,Z 71.369,A 49.843,B 90.000,C 0.000} C_DIS
LIN {X -186.704,Y -221.904,Z 71.092,A 49.924,B 90.000,C 0.000} C_DIS
LIN {X -186.418,Y -222.145,Z 70.970,A 49.998,B 90.000,C 0.000} C_DIS
LIN {X -186.093,Y -222.417,Z 70.982,A 50.081,B 90.000,C 0.000} C_DIS
LIN {X -185.826,Y -222.640,Z 71.160,A 50.150,B 90.000,C 0.000} C_DIS
LIN {X -185.625,Y -222.808,Z 71.495,A 50.202,B 90.000,C 0.000} C_DIS
LIN {X -185.499,Y -222.913,Z 71.975,A 50.234,B 90.000,C 0.000} C_DIS
LIN {X -185.287,Y -223.089,Z 74.107,A 50.289,B 90.000,C 0.000} C_DIS
LIN {X -185.083,Y -223.259,Z 74.592,A 50.341,B 90.000,C 0.000} C_DIS
LIN {X -184.778,Y -223.510,Z 74.852,A 50.419,B 90.000,C 0.000} C_DIS
LIN {X -183.947,Y -224.196,Z 75.006,A 50.632,B 90.000,C 0.000} C_DIS
LIN {X -183.990,Y -224.160,Z 74.699,A 50.621,B 90.000,C 0.000} C_DIS
LIN {X -183.997,Y -224.154,Z 73.772,A 50.619,B 90.000,C 0.000} C_DIS
LIN {X -183.610,Y -224.472,Z 71.323,A 50.718,B 90.000,C 0.000} C_DIS
LIN {X -183.527,Y -224.539,Z 70.813,A 50.739,B 90.000,C 0.000} C_DIS
LIN {X -183.472,Y -224.584,Z 69.582,A 50.753,B 90.000,C 0.000} C_DIS
LIN {X -183.625,Y -224.459,Z 68.611,A 50.714,B 90.000,C 0.000} C_DIS
LIN {X -183.988,Y -224.161,Z 67.804,A 50.621,B 90.000,C 0.000} C_DIS
LIN {X -184.449,Y -223.782,Z 67.188,A 50.503,B 90.000,C 0.000} C_DIS
LIN {X -185.965,Y -222.524,Z 65.648,A 50.114,B 90.000,C 0.000} C_DIS
LIN {X -187.247,Y -221.446,Z 63.793,A 49.783,B 90.000,C 0.000} C_DIS
LIN {X -187.530,Y -221.207,Z 63.270,A 49.710,B 90.000,C 0.000} C_DIS
LIN {X -188.028,Y -220.784,Z 62.101,A 49.581,B 90.000,C 0.000} C_DIS
LIN {X -188.336,Y -220.521,Z 60.990,A 49.501,B 90.000,C 0.000} C_DIS
LIN {X -188.454,Y -220.420,Z 59.945,A 49.470,B 90.000,C 0.000} C_DIS
LIN {X -188.381,Y -220.482,Z 58.974,A 49.489,B 90.000,C 0.000} C_DIS
LIN {X -188.178,Y -220.656,Z 58.234,A 49.542,B 90.000,C 0.000} C_DIS
LIN {X -187.856,Y -220.930,Z 57.518,A 49.626,B 90.000,C 0.000} C_DIS
LIN {X -187.446,Y -221.278,Z 56.885,A 49.732,B 90.000,C 0.000} C_DIS
LIN {X -186.979,Y -221.673,Z 56.393,A 49.853,B 90.000,C 0.000} C_DIS
LIN {X -186.437,Y -222.129,Z 56.042,A 49.993,B 90.000,C 0.000} C_DIS
LIN {X -185.844,Y -222.626,Z 55.797,A 50.146,B 90.000,C 0.000} C_DIS
LIN {X -185.844,Y -222.626,Z 55.797,A 50.146,B 90.000,C 0.000} C_DIS
LIN {X -185.479,Y -222.930,Z 55.712,A 50.239,B 90.000,C 0.000} C_DIS
LIN {X -185.451,Y -222.953,Z 55.802,A 50.246,B 90.000,C 0.000} C_DIS
LIN {X -185.733,Y -222.718,Z 57.217,A 50.174,B 90.000,C 0.000} C_DIS
LIN {X -185.717,Y -222.731,Z 58.352,A 50.178,B 90.000,C 0.000} C_DIS
LIN {X -185.432,Y -222.968,Z 59.432,A 50.251,B 90.000,C 0.000} C_DIS
LIN {X -184.871,Y -223.434,Z 60.475,A 50.395,B 90.000,C 0.000} C_DIS
LIN {X -184.024,Y -224.132,Z 61.501,A 50.612,B 90.000,C 0.000} C_DIS
LIN {X -182.455,Y -225.410,Z 62.970,A 51.012,B 90.000,C 0.000} C_DIS
LIN {X -181.574,Y -226.122,Z 63.815,A 51.236,B 90.000,C 0.000} C_DIS
LIN {X -180.007,Y -227.370,Z 62.320,A 51.632,B 90.000,C 0.000} C_DIS
LIN {X -178.536,Y -228.528,Z 60.759,A 52.001,B 90.000,C 0.000} C_DIS
LIN {X -178.074,Y -228.887,Z 60.095,A 52.117,B 90.000,C 0.000} C_DIS
LIN {X -177.738,Y -229.149,Z 59.453,A 52.201,B 90.000,C 0.000} C_DIS
LIN {X -177.500,Y -229.334,Z 58.782,A 52.261,B 90.000,C 0.000} C_DIS
LIN {X -177.391,Y -229.418,Z 58.033,A 52.288,B 90.000,C 0.000} C_DIS
LIN {X -177.388,Y -229.420,Z 57.096,A 52.289,B 90.000,C 0.000} C_DIS
LIN {X -177.548,Y -229.296,Z 56.326,A 52.249,B 90.000,C 0.000} C_DIS
LIN {X -177.691,Y -229.185,Z 55.853,A 52.213,B 90.000,C 0.000} C_DIS
LIN {X -177.722,Y -229.161,Z 55.690,A 52.205,B 90.000,C 0.000} C_DIS
LIN {X -176.963,Y -229.748,Z 55.874,A 52.395,B 90.000,C 0.000} C_DIS
LIN {X -176.472,Y -230.125,Z 56.128,A 52.517,B 90.000,C 0.000} C_DIS
LIN {X -176.010,Y -230.479,Z 56.489,A 52.632,B 90.000,C 0.000} C_DIS
LIN {X -175.582,Y -230.805,Z 56.955,A 52.738,B 90.000,C 0.000} C_DIS
LIN {X -175.219,Y -231.081,Z 57.467,A 52.829,B 90.000,C 0.000} C_DIS
LIN {X -174.962,Y -231.275,Z 58.042,A 52.892,B 90.000,C 0.000} C_DIS
LIN {X -174.673,Y -231.494,Z 59.021,A 52.964,B 90.000,C 0.000} C_DIS
LIN {X -174.592,Y -231.555,Z 60.038,A 52.984,B 90.000,C 0.000} C_DIS
LIN {X -174.640,Y -231.519,Z 60.810,A 52.972,B 90.000,C 0.000} C_DIS
LIN {X -174.795,Y -231.402,Z 61.558,A 52.934,B 90.000,C 0.000} C_DIS
LIN {X -175.072,Y -231.192,Z 62.340,A 52.865,B 90.000,C 0.000} C_DIS
LIN {X -176.196,Y -230.337,Z 64.402,A 52.586,B 90.000,C 0.000} C_DIS
LIN {X -177.635,Y -229.228,Z 66.120,A 52.227,B 90.000,C 0.000} C_DIS
LIN {X -178.755,Y -228.356,Z 67.257,A 51.946,B 90.000,C 0.000} C_DIS
LIN {X -179.265,Y -227.956,Z 67.976,A 51.818,B 90.000,C 0.000} C_DIS
LIN {X -179.474,Y -227.792,Z 68.389,A 51.766,B 90.000,C 0.000} C_DIS
LIN {X -179.593,Y -227.698,Z 68.780,A 51.736,B 90.000,C 0.000} C_DIS
LIN {X -179.635,Y -227.665,Z 70.945,A 51.725,B 90.000,C 0.000} C_DIS
LIN {X -179.227,Y -227.986,Z 73.345,A 51.828,B 90.000,C 0.000} C_DIS
LIN {X -179.176,Y -228.026,Z 75.006,A 51.841,B 90.000,C 0.000} C_DIS
LIN {X -178.394,Y -228.638,Z 74.862,A 52.037,B 90.000,C 0.000} C_DIS
LIN {X -178.097,Y -228.870,Z 74.614,A 52.111,B 90.000,C 0.000} C_DIS
LIN {X -177.887,Y -229.033,Z 74.163,A 52.164,B 90.000,C 0.000} C_DIS
LIN {X -177.656,Y -229.213,Z 72.148,A 52.222,B 90.000,C 0.000} C_DIS
LIN {X -177.457,Y -229.366,Z 71.449,A 52.271,B 90.000,C 0.000} C_DIS
LIN {X -177.196,Y -229.568,Z 71.056,A 52.337,B 90.000,C 0.000} C_DIS
LIN {X -176.809,Y -229.867,Z 70.964,A 52.433,B 90.000,C 0.000} C_DIS
LIN {X -176.319,Y -230.242,Z 71.140,A 52.555,B 90.000,C 0.000} C_DIS
LIN {X -175.822,Y -230.622,Z 71.627,A 52.679,B 90.000,C 0.000} C_DIS
LIN {X -174.561,Y -231.578,Z 73.562,A 52.991,B 90.000,C 0.000} C_DIS
LIN {X -174.148,Y -231.889,Z 74.416,A 53.094,B 90.000,C 0.000} C_DIS
LIN {X -173.590,Y -232.307,Z 76.166,A 53.231,B 90.000,C 0.000} C_DIS
LIN {X -173.477,Y -232.391,Z 76.357,A 53.259,B 90.000,C 0.000} C_DIS
LIN {X -173.360,Y -232.478,Z 76.413,A 53.288,B 90.000,C 0.000} C_DIS
LIN {X -173.189,Y -232.606,Z 76.238,A 53.330,B 90.000,C 0.000} C_DIS
LIN {X -173.115,Y -232.661,Z 75.743,A 53.348,B 90.000,C 0.000} C_DIS
LIN {X -173.140,Y -232.642,Z 74.971,A 53.342,B 90.000,C 0.000} C_DIS
LIN {X -173.489,Y -232.383,Z 72.734,A 53.256,B 90.000,C 0.000} C_DIS
LIN {X -173.743,Y -232.192,Z 71.932,A 53.193,B 90.000,C 0.000} C_DIS
LIN {X -174.148,Y -231.889,Z 71.308,A 53.094,B 90.000,C 0.000} C_DIS
LIN {X -175.585,Y -230.803,Z 69.776,A 52.738,B 90.000,C 0.000} C_DIS
LIN {X -175.966,Y -230.513,Z 69.086,A 52.643,B 90.000,C 0.000} C_DIS
LIN {X -176.084,Y -230.422,Z 68.690,A 52.614,B 90.000,C 0.000} C_DIS
LIN {X -176.110,Y -230.403,Z 68.247,A 52.607,B 90.000,C 0.000} C_DIS
LIN {X -176.084,Y -230.422,Z 67.802,A 52.614,B 90.000,C 0.000} C_DIS
LIN {X -175.958,Y -230.518,Z 67.404,A 52.645,B 90.000,C 0.000} C_DIS
LIN {X -175.462,Y -230.897,Z 66.449,A 52.768,B 90.000,C 0.000} C_DIS
LIN {X -173.969,Y -232.023,Z 64.790,A 53.138,B 90.000,C 0.000} C_DIS
LIN {X -173.664,Y -232.252,Z 64.460,A 53.213,B 90.000,C 0.000} C_DIS
LIN {X -172.856,Y -232.854,Z 63.314,A 53.412,B 90.000,C 0.000} C_DIS
LIN {X -172.374,Y -233.211,Z 62.262,A 53.531,B 90.000,C 0.000} C_DIS
LIN {X -172.051,Y -233.449,Z 61.180,A 53.610,B 90.000,C 0.000} C_DIS
LIN {X -171.954,Y -233.520,Z 60.594,A 53.634,B 90.000,C 0.000} C_DIS
LIN {X -171.949,Y -233.524,Z 59.244,A 53.635,B 90.000,C 0.000} C_DIS
LIN {X -172.054,Y -233.447,Z 58.747,A 53.609,B 90.000,C 0.000} C_DIS
LIN {X -172.342,Y -233.234,Z 57.992,A 53.538,B 90.000,C 0.000} C_DIS
LIN {X -173.161,Y -232.627,Z 56.938,A 53.337,B 90.000,C 0.000} C_DIS
LIN {X -173.341,Y -232.493,Z 56.433,A 53.293,B 90.000,C 0.000} C_DIS
LIN {X -173.329,Y -232.502,Z 56.293,A 53.296,B 90.000,C 0.000} C_DIS
LIN {X -173.104,Y -232.669,Z 56.213,A 53.351,B 90.000,C 0.000} C_DIS
LIN {X -172.691,Y -232.976,Z 56.173,A 53.453,B 90.000,C 0.000} C_DIS
LIN {X -172.215,Y -233.328,Z 56.254,A 53.570,B 90.000,C 0.000} C_DIS
LIN {X -171.029,Y -234.199,Z 56.792,A 53.860,B 90.000,C 0.000} C_DIS
LIN {X -169.323,Y -235.435,Z 58.136,A 54.277,B 90.000,C 0.000} C_DIS
LIN {X -167.788,Y -236.531,Z 59.778,A 54.649,B 90.000,C 0.000} C_DIS
LIN {X -167.432,Y -236.784,Z 60.213,A 54.735,B 90.000,C 0.000} C_DIS
LIN {X -166.765,Y -237.254,Z 61.293,A 54.897,B 90.000,C 0.000} C_DIS
LIN {X -165.758,Y -237.958,Z 63.469,A 55.140,B 90.000,C 0.000} C_DIS
LIN {X -164.747,Y -238.659,Z 65.645,A 55.383,B 90.000,C 0.000} C_DIS
LIN {X -163.697,Y -239.377,Z 67.798,A 55.634,B 90.000,C 0.000} C_DIS
LIN {X -162.636,Y -240.099,Z 69.943,A 55.887,B 90.000,C 0.000} C_DIS
LIN {X -161.538,Y -240.842,Z 72.063,A 56.149,B 90.000,C 0.000} C_DIS
LIN {X -160.352,Y -241.633,Z 74.116,A 56.431,B 90.000,C 0.000} C_DIS
LIN {X -159.100,Y -242.457,Z 76.117,A 56.727,B 90.000,C 0.000} C_DIS
LIN {X -157.811,Y -243.298,Z 78.087,A 57.031,B 90.000,C 0.000} C_DIS
LIN {X -156.520,Y -244.130,Z 80.060,A 57.335,B 90.000,C 0.000} C_DIS
LIN {X -155.227,Y -244.949,Z 82.036,A 57.637,B 90.000,C 0.000} C_DIS
LIN {X -153.934,Y -245.769,Z 84.012,A 57.940,B 90.000,C 0.000} C_DIS
LIN {X -152.702,Y -246.540,Z 86.046,A 58.227,B 90.000,C 0.000} C_DIS
LIN {X -151.714,Y -247.149,Z 88.261,A 58.456,B 90.000,C 0.000} C_DIS
LIN {X -151.071,Y -247.543,Z 90.644,A 58.605,B 90.000,C 0.000} C_DIS
LIN {X -150.609,Y -247.824,Z 93.085,A 58.712,B 90.000,C 0.000} C_DIS
LIN {X -150.170,Y -248.090,Z 95.531,A 58.813,B 90.000,C 0.000} C_DIS
LIN {X -149.778,Y -248.327,Z 97.989,A 58.904,B 90.000,C 0.000} C_DIS
LIN {X -149.399,Y -248.555,Z 100.449,A 58.991,B 90.000,C 0.000} C_DIS
LIN {X -149.082,Y -248.746,Z 102.922,A 59.064,B 90.000,C 0.000} C_DIS
LIN {X -148.760,Y -248.939,Z 105.394,A 59.138,B 90.000,C 0.000} C_DIS
LIN {X -148.353,Y -249.181,Z 107.848,A 59.232,B 90.000,C 0.000} C_DIS
LIN {X -148.309,Y -249.208,Z 108.080,A 59.242,B 90.000,C 0.000} C_DIS
LIN {X -147.948,Y -249.422,Z 109.280,A 59.325,B 90.000,C 0.000} C_DIS
LIN {X -147.495,Y -249.690,Z 110.261,A 59.429,B 90.000,C 0.000} C_DIS
LIN {X -147.268,Y -249.824,Z 110.608,A 59.481,B 90.000,C 0.000} C_DIS
LIN {X -147.028,Y -249.965,Z 110.803,A 59.536,B 90.000,C 0.000} C_DIS
LIN {X -144.983,Y -251.157,Z 111.606,A 60.004,B 90.000,C 0.000} C_DIS
LIN {X -143.847,Y -251.810,Z 112.004,A 60.263,B 90.000,C 0.000} C_DIS
LIN {X -142.512,Y -252.567,Z 112.758,A 60.566,B 90.000,C 0.000} C_DIS
LIN {X -141.282,Y -253.258,Z 113.708,A 60.845,B 90.000,C 0.000} C_DIS
LIN {X -140.641,Y -253.614,Z 114.461,A 60.989,B 90.000,C 0.000} C_DIS
LIN {X -140.094,Y -253.917,Z 115.436,A 61.113,B 90.000,C 0.000} C_DIS
LIN {X -139.616,Y -254.180,Z 116.686,A 61.221,B 90.000,C 0.000} C_DIS
LIN {X -139.028,Y -254.502,Z 119.095,A 61.353,B 90.000,C 0.000} C_DIS
LIN {X -138.820,Y -254.615,Z 120.208,A 61.400,B 90.000,C 0.000} C_DIS
LIN {X -138.714,Y -254.673,Z 122.705,A 61.424,B 90.000,C 0.000} C_DIS
LIN {X -138.617,Y -254.726,Z 125.203,A 61.446,B 90.000,C 0.000} C_DIS
LIN {X -138.614,Y -254.727,Z 125.264,A 61.446,B 90.000,C 0.000} C_DIS
LIN {X -138.227,Y -254.938,Z 127.725,A 61.533,B 90.000,C 0.000} C_DIS
LIN {X -137.979,Y -255.072,Z 128.834,A 61.589,B 90.000,C 0.000} C_DIS
LIN {X -137.172,Y -255.507,Z 131.160,A 61.770,B 90.000,C 0.000} C_DIS
LIN {X -136.741,Y -255.738,Z 132.605,A 61.867,B 90.000,C 0.000} C_DIS
LIN {X -136.629,Y -255.798,Z 133.404,A 61.892,B 90.000,C 0.000} C_DIS
LIN {X -136.620,Y -255.802,Z 134.191,A 61.894,B 90.000,C 0.000} C_DIS
LIN {X -136.754,Y -255.731,Z 135.162,A 61.864,B 90.000,C 0.000} C_DIS
LIN {X -137.571,Y -255.292,Z 137.484,A 61.681,B 90.000,C 0.000} C_DIS
LIN {X -138.346,Y -254.873,Z 139.823,A 61.507,B 90.000,C 0.000} C_DIS
LIN {X -138.373,Y -254.858,Z 139.897,A 61.501,B 90.000,C 0.000} C_DIS
LIN {X -138.553,Y -254.761,Z 140.016,A 61.460,B 90.000,C 0.000} C_DIS
LIN {X -138.809,Y -254.621,Z 140.067,A 61.403,B 90.000,C 0.000} C_DIS
LIN {X -139.490,Y -254.249,Z 139.981,A 61.249,B 90.000,C 0.000} C_DIS
LIN {X -140.285,Y -253.811,Z 139.674,A 61.070,B 90.000,C 0.000} C_DIS
LIN {X -141.068,Y -253.377,Z 139.180,A 60.893,B 90.000,C 0.000} C_DIS
LIN {X -141.860,Y -252.934,Z 138.418,A 60.714,B 90.000,C 0.000} C_DIS
LIN {X -143.295,Y -252.124,Z 136.538,A 60.388,B 90.000,C 0.000} C_DIS
LIN {X -144.531,Y -251.417,Z 134.483,A 60.107,B 90.000,C 0.000} C_DIS
LIN {X -145.253,Y -251.001,Z 133.195,A 59.942,B 90.000,C 0.000} C_DIS
LIN {X -145.496,Y -250.860,Z 133.931,A 59.887,B 90.000,C 0.000} C_DIS
LIN {X -145.933,Y -250.606,Z 136.379,A 59.787,B 90.000,C 0.000} C_DIS
LIN {X -146.050,Y -250.538,Z 137.298,A 59.760,B 90.000,C 0.000} C_DIS
LIN {X -146.111,Y -250.503,Z 139.797,A 59.746,B 90.000,C 0.000} C_DIS
LIN {X -146.053,Y -250.537,Z 142.296,A 59.760,B 90.000,C 0.000} C_DIS
LIN {X -145.812,Y -250.677,Z 144.780,A 59.815,B 90.000,C 0.000} C_DIS
LIN {X -145.413,Y -250.908,Z 147.094,A 59.906,B 90.000,C 0.000} C_DIS
LIN {X -145.146,Y -251.063,Z 147.988,A 59.967,B 90.000,C 0.000} C_DIS
LIN {X -143.970,Y -251.739,Z 146.870,A 60.235,B 90.000,C 0.000} C_DIS
LIN {X -143.403,Y -252.063,Z 146.709,A 60.364,B 90.000,C 0.000} C_DIS
LIN {X -142.956,Y -252.316,Z 146.786,A 60.465,B 90.000,C 0.000} C_DIS
LIN {X -142.603,Y -252.516,Z 147.032,A 60.545,B 90.000,C 0.000} C_DIS
LIN {X -142.324,Y -252.674,Z 147.467,A 60.609,B 90.000,C 0.000} C_DIS
LIN {X -142.099,Y -252.800,Z 148.113,A 60.660,B 90.000,C 0.000} C_DIS
LIN {X -141.906,Y -252.908,Z 149.255,A 60.703,B 90.000,C 0.000} C_DIS
LIN {X -141.770,Y -252.985,Z 151.751,A 60.734,B 90.000,C 0.000} C_DIS
LIN {X -141.679,Y -253.036,Z 154.248,A 60.755,B 90.000,C 0.000} C_DIS
LIN {X -141.641,Y -253.057,Z 156.748,A 60.763,B 90.000,C 0.000} C_DIS
LIN {X -141.611,Y -253.074,Z 159.248,A 60.770,B 90.000,C 0.000} C_DIS
LIN {X -141.677,Y -253.037,Z 161.746,A 60.755,B 90.000,C 0.000} C_DIS
LIN {X -141.756,Y -252.993,Z 164.245,A 60.737,B 90.000,C 0.000} C_DIS
LIN {X -141.941,Y -252.889,Z 166.735,A 60.696,B 90.000,C 0.000} C_DIS
LIN {X -142.352,Y -252.658,Z 169.190,A 60.602,B 90.000,C 0.000} C_DIS
LIN {X -142.894,Y -252.352,Z 171.088,A 60.479,B 90.000,C 0.000} C_DIS
LIN {X -143.168,Y -252.196,Z 171.728,A 60.417,B 90.000,C 0.000} C_DIS
LIN {X -143.459,Y -252.031,Z 172.113,A 60.351,B 90.000,C 0.000} C_DIS
LIN {X -143.760,Y -251.859,Z 172.234,A 60.282,B 90.000,C 0.000} C_DIS
LIN {X -144.061,Y -251.687,Z 172.083,A 60.214,B 90.000,C 0.000} C_DIS
LIN {X -144.258,Y -251.574,Z 171.782,A 60.169,B 90.000,C 0.000} C_DIS
LIN {X -144.384,Y -251.502,Z 171.250,A 60.140,B 90.000,C 0.000} C_DIS
LIN {X -144.499,Y -251.436,Z 168.754,A 60.114,B 90.000,C 0.000} C_DIS
LIN {X -144.506,Y -251.432,Z 167.435,A 60.113,B 90.000,C 0.000} C_DIS
LIN {X -144.337,Y -251.529,Z 165.568,A 60.151,B 90.000,C 0.000} C_DIS
LIN {X -144.562,Y -251.400,Z 163.082,A 60.100,B 90.000,C 0.000} C_DIS
LIN {X -144.792,Y -251.267,Z 160.596,A 60.047,B 90.000,C 0.000} C_DIS
LIN {X -145.143,Y -251.065,Z 158.129,A 59.967,B 90.000,C 0.000} C_DIS
LIN {X -145.630,Y -250.782,Z 155.693,A 59.856,B 90.000,C 0.000} C_DIS
LIN {X -145.683,Y -250.752,Z 155.438,A 59.844,B 90.000,C 0.000} C_DIS
LIN {X -146.468,Y -250.292,Z 153.109,A 59.664,B 90.000,C 0.000} C_DIS
LIN {X -147.365,Y -249.760,Z 150.837,A 59.458,B 90.000,C 0.000} C_DIS
LIN {X -148.262,Y -249.229,Z 148.565,A 59.252,B 90.000,C 0.000} C_DIS
LIN {X -149.159,Y -248.697,Z 146.293,A 59.046,B 90.000,C 0.000} C_DIS
LIN {X -149.942,Y -248.229,Z 144.217,A 58.866,B 90.000,C 0.000} C_DIS
LIN {X -150.264,Y -248.034,Z 142.929,A 58.792,B 90.000,C 0.000} C_DIS
LIN {X -150.412,Y -247.944,Z 141.672,A 58.757,B 90.000,C 0.000} C_DIS
LIN {X -150.284,Y -248.022,Z 139.177,A 58.787,B 90.000,C 0.000} C_DIS
LIN {X -149.896,Y -248.256,Z 136.718,A 58.877,B 90.000,C 0.000} C_DIS
LIN {X -149.370,Y -248.572,Z 134.295,A 58.998,B 90.000,C 0.000} C_DIS
LIN {X -148.831,Y -248.896,Z 131.875,A 59.122,B 90.000,C 0.000} C_DIS
LIN {X -148.267,Y -249.232,Z 129.463,A 59.252,B 90.000,C 0.000} C_DIS
LIN {X -147.790,Y -249.516,Z 127.025,A 59.361,B 90.000,C 0.000} C_DIS
LIN {X -147.552,Y -249.657,Z 124.541,A 59.416,B 90.000,C 0.000} C_DIS
LIN {X -147.556,Y -249.654,Z 122.225,A 59.415,B 90.000,C 0.000} C_DIS
LIN {X -147.898,Y -249.452,Z 119.756,A 59.337,B 90.000,C 0.000} C_DIS
LIN {X -148.340,Y -249.189,Z 117.310,A 59.235,B 90.000,C 0.000} C_DIS
LIN {X -148.918,Y -248.844,Z 114.902,A 59.102,B 90.000,C 0.000} C_DIS
LIN {X -149.391,Y -248.560,Z 113.226,A 58.993,B 90.000,C 0.000} C_DIS
LIN {X -149.601,Y -248.434,Z 112.901,A 58.945,B 90.000,C 0.000} C_DIS
LIN {X -149.887,Y -248.262,Z 112.665,A 58.879,B 90.000,C 0.000} C_DIS
LIN {X -150.260,Y -248.036,Z 112.505,A 58.793,B 90.000,C 0.000} C_DIS
LIN {X -150.965,Y -247.608,Z 112.441,A 58.630,B 90.000,C 0.000} C_DIS
LIN {X -151.602,Y -247.218,Z 112.656,A 58.482,B 90.000,C 0.000} C_DIS
LIN {X -152.295,Y -246.792,Z 113.267,A 58.321,B 90.000,C 0.000} C_DIS
LIN {X -152.846,Y -246.451,Z 114.139,A 58.193,B 90.000,C 0.000} C_DIS
LIN {X -153.254,Y -246.198,Z 115.272,A 58.098,B 90.000,C 0.000} C_DIS
LIN {X -153.517,Y -246.034,Z 116.661,A 58.037,B 90.000,C 0.000} C_DIS
LIN {X -153.641,Y -245.956,Z 119.157,A 58.008,B 90.000,C 0.000} C_DIS
LIN {X -153.735,Y -245.897,Z 121.048,A 57.986,B 90.000,C 0.000} C_DIS
LIN {X -153.668,Y -245.939,Z 122.392,A 58.002,B 90.000,C 0.000} C_DIS
LIN {X -153.214,Y -246.222,Z 123.804,A 58.108,B 90.000,C 0.000} C_DIS
LIN {X -153.161,Y -246.255,Z 124.145,A 58.120,B 90.000,C 0.000} C_DIS
LIN {X -153.235,Y -246.209,Z 124.451,A 58.103,B 90.000,C 0.000} C_DIS
LIN {X -153.438,Y -246.083,Z 124.818,A 58.056,B 90.000,C 0.000} C_DIS
LIN {X -153.702,Y -245.918,Z 125.175,A 57.994,B 90.000,C 0.000} C_DIS
LIN {X -154.059,Y -245.694,Z 125.362,A 57.911,B 90.000,C 0.000} C_DIS
LIN {X -154.837,Y -245.205,Z 125.609,A 57.729,B 90.000,C 0.000} C_DIS
LIN {X -155.599,Y -244.722,Z 125.684,A 57.551,B 90.000,C 0.000} C_DIS
LIN {X -156.296,Y -244.278,Z 125.626,A 57.388,B 90.000,C 0.000} C_DIS
LIN {X -156.859,Y -243.916,Z 125.418,A 57.255,B 90.000,C 0.000} C_DIS
LIN {X -157.209,Y -243.691,Z 125.139,A 57.173,B 90.000,C 0.000} C_DIS
LIN {X -158.471,Y -242.872,Z 123.689,A 56.876,B 90.000,C 0.000} C_DIS
LIN {X -159.028,Y -242.508,Z 123.186,A 56.745,B 90.000,C 0.000} C_DIS
LIN {X -160.883,Y -241.281,Z 122.044,A 56.305,B 90.000,C 0.000} C_DIS
LIN {X -161.496,Y -240.871,Z 121.749,A 56.159,B 90.000,C 0.000} C_DIS
LIN {X -162.356,Y -240.293,Z 119.608,A 55.955,B 90.000,C 0.000} C_DIS
LIN {X -162.452,Y -240.227,Z 119.005,A 55.932,B 90.000,C 0.000} C_DIS
LIN {X -162.477,Y -240.211,Z 118.288,A 55.926,B 90.000,C 0.000} C_DIS
LIN {X -162.324,Y -240.314,Z 116.575,A 55.962,B 90.000,C 0.000} C_DIS
LIN {X -162.148,Y -240.433,Z 115.778,A 56.004,B 90.000,C 0.000} C_DIS
LIN {X -161.919,Y -240.587,Z 115.102,A 56.059,B 90.000,C 0.000} C_DIS
LIN {X -161.627,Y -240.784,Z 114.641,A 56.128,B 90.000,C 0.000} C_DIS
LIN {X -159.942,Y -241.905,Z 113.174,A 56.528,B 90.000,C 0.000} C_DIS
LIN {X -158.459,Y -242.880,Z 112.143,A 56.879,B 90.000,C 0.000} C_DIS
LIN {X -157.586,Y -243.447,Z 111.726,A 57.085,B 90.000,C 0.000} C_DIS
LIN {X -155.506,Y -244.781,Z 111.351,A 57.573,B 90.000,C 0.000} C_DIS
LIN {X -155.395,Y -244.852,Z 111.328,A 57.599,B 90.000,C 0.000} C_DIS
LIN {X -155.010,Y -245.096,Z 111.151,A 57.689,B 90.000,C 0.000} C_DIS
LIN {X -154.586,Y -245.363,Z 110.844,A 57.788,B 90.000,C 0.000} C_DIS
LIN {X -154.529,Y -245.399,Z 110.698,A 57.801,B 90.000,C 0.000} C_DIS
LIN {X -154.605,Y -245.352,Z 110.372,A 57.784,B 90.000,C 0.000} C_DIS
LIN {X -154.807,Y -245.224,Z 109.830,A 57.736,B 90.000,C 0.000} C_DIS
LIN {X -155.096,Y -245.041,Z 109.315,A 57.669,B 90.000,C 0.000} C_DIS
LIN {X -155.459,Y -244.811,Z 108.845,A 57.584,B 90.000,C 0.000} C_DIS
LIN {X -155.885,Y -244.540,Z 108.438,A 57.484,B 90.000,C 0.000} C_DIS
LIN {X -157.024,Y -243.810,Z 107.764,A 57.217,B 90.000,C 0.000} C_DIS
LIN {X -159.007,Y -242.521,Z 106.954,A 56.749,B 90.000,C 0.000} C_DIS
LIN {X -159.958,Y -241.896,Z 106.539,A 56.525,B 90.000,C 0.000} C_DIS
LIN {X -160.290,Y -241.675,Z 106.291,A 56.446,B 90.000,C 0.000} C_DIS
LIN {X -160.634,Y -241.447,Z 105.830,A 56.364,B 90.000,C 0.000} C_DIS
LIN {X -161.740,Y -240.707,Z 103.714,A 56.101,B 90.000,C 0.000} C_DIS
LIN {X -162.812,Y -239.983,Z 101.575,A 55.846,B 90.000,C 0.000} C_DIS
LIN {X -163.801,Y -239.310,Z 99.380,A 55.610,B 90.000,C 0.000} C_DIS
LIN {X -163.838,Y -239.284,Z 99.290,A 55.600,B 90.000,C 0.000} C_DIS
LIN {X -164.010,Y -239.167,Z 99.057,A 55.559,B 90.000,C 0.000} C_DIS
LIN {X -164.096,Y -239.107,Z 99.242,A 55.539,B 90.000,C 0.000} C_DIS
LIN {X -164.783,Y -238.633,Z 101.599,A 55.374,B 90.000,C 0.000} C_DIS
LIN {X -165.500,Y -238.138,Z 103.942,A 55.202,B 90.000,C 0.000} C_DIS
LIN {X -166.419,Y -237.497,Z 106.177,A 54.980,B 90.000,C 0.000} C_DIS
LIN {X -167.452,Y -236.769,Z 108.334,A 54.731,B 90.000,C 0.000} C_DIS
LIN {X -168.612,Y -235.945,Z 110.389,A 54.450,B 90.000,C 0.000} C_DIS
LIN {X -168.939,Y -235.711,Z 110.835,A 54.370,B 90.000,C 0.000} C_DIS
LIN {X -169.850,Y -235.055,Z 111.829,A 54.148,B 90.000,C 0.000} C_DIS
LIN {X -170.803,Y -234.364,Z 112.537,A 53.916,B 90.000,C 0.000} C_DIS
LIN {X -171.810,Y -233.627,Z 112.965,A 53.669,B 90.000,C 0.000} C_DIS
LIN {X -172.884,Y -232.833,Z 113.123,A 53.405,B 90.000,C 0.000} C_DIS
LIN {X -173.391,Y -232.455,Z 113.096,A 53.280,B 90.000,C 0.000} C_DIS
LIN {X -173.772,Y -232.171,Z 112.959,A 53.186,B 90.000,C 0.000} C_DIS
LIN {X -174.101,Y -231.924,Z 112.666,A 53.105,B 90.000,C 0.000} C_DIS
LIN {X -174.453,Y -231.660,Z 112.172,A 53.018,B 90.000,C 0.000} C_DIS
LIN {X -174.826,Y -231.379,Z 111.430,A 52.926,B 90.000,C 0.000} C_DIS
LIN {X -175.020,Y -231.232,Z 110.595,A 52.878,B 90.000,C 0.000} C_DIS
LIN {X -175.023,Y -231.229,Z 110.404,A 52.877,B 90.000,C 0.000} C_DIS
LIN {X -174.913,Y -231.313,Z 110.296,A 52.904,B 90.000,C 0.000} C_DIS
LIN {X -173.626,Y -232.280,Z 109.917,A 53.223,B 90.000,C 0.000} C_DIS
LIN {X -173.100,Y -232.672,Z 109.643,A 53.352,B 90.000,C 0.000} C_DIS
LIN {X -172.593,Y -233.049,Z 109.235,A 53.477,B 90.000,C 0.000} C_DIS
LIN {X -171.100,Y -234.147,Z 107.557,A 53.843,B 90.000,C 0.000} C_DIS
LIN {X -170.963,Y -234.247,Z 107.385,A 53.877,B 90.000,C 0.000} C_DIS
LIN {X -170.002,Y -234.945,Z 105.299,A 54.111,B 90.000,C 0.000} C_DIS
LIN {X -169.830,Y -235.070,Z 104.703,A 54.153,B 90.000,C 0.000} C_DIS
LIN {X -169.478,Y -235.324,Z 102.241,A 54.239,B 90.000,C 0.000} C_DIS
LIN {X -169.253,Y -235.485,Z 100.663,A 54.294,B 90.000,C 0.000} C_DIS
LIN {X -169.046,Y -235.634,Z 99.908,A 54.344,B 90.000,C 0.000} C_DIS
LIN {X -168.738,Y -235.854,Z 99.156,A 54.419,B 90.000,C 0.000} C_DIS
LIN {X -167.535,Y -236.710,Z 97.139,A 54.711,B 90.000,C 0.000} C_DIS
LIN {X -166.302,Y -237.579,Z 95.145,A 55.009,B 90.000,C 0.000} C_DIS
LIN {X -166.284,Y -237.591,Z 95.117,A 55.013,B 90.000,C 0.000} C_DIS
LIN {X -165.315,Y -238.267,Z 92.914,A 55.246,B 90.000,C 0.000} C_DIS
LIN {X -164.840,Y -238.595,Z 91.836,A 55.360,B 90.000,C 0.000} C_DIS
LIN {X -164.636,Y -238.736,Z 91.645,A 55.409,B 90.000,C 0.000} C_DIS
LIN {X -164.402,Y -238.898,Z 91.620,A 55.465,B 90.000,C 0.000} C_DIS
LIN {X -164.106,Y -239.101,Z 91.731,A 55.536,B 90.000,C 0.000} C_DIS
LIN {X -163.810,Y -239.304,Z 92.036,A 55.607,B 90.000,C 0.000} C_DIS
LIN {X -162.662,Y -240.085,Z 94.115,A 55.882,B 90.000,C 0.000} C_DIS
LIN {X -161.479,Y -240.879,Z 96.169,A 56.163,B 90.000,C 0.000} C_DIS
LIN {X -160.240,Y -241.701,Z 98.178,A 56.457,B 90.000,C 0.000} C_DIS
LIN {X -159.001,Y -242.523,Z 100.188,A 56.751,B 90.000,C 0.000} C_DIS
LIN {X -157.748,Y -243.341,Z 102.191,A 57.046,B 90.000,C 0.000} C_DIS
LIN {X -156.434,Y -244.189,Z 104.141,A 57.355,B 90.000,C 0.000} C_DIS
LIN {X -156.351,Y -244.243,Z 104.259,A 57.375,B 90.000,C 0.000} C_DIS
LIN {X -155.169,Y -244.995,Z 105.581,A 57.652,B 90.000,C 0.000} C_DIS
LIN {X -153.832,Y -245.836,Z 106.666,A 57.964,B 90.000,C 0.000} C_DIS
LIN {X -152.654,Y -246.570,Z 107.283,A 58.238,B 90.000,C 0.000} C_DIS
LIN {X -152.514,Y -246.657,Z 107.324,A 58.270,B 90.000,C 0.000} C_DIS
LIN {X -152.624,Y -246.588,Z 107.093,A 58.245,B 90.000,C 0.000} C_DIS
LIN {X -153.884,Y -245.804,Z 105.080,A 57.952,B 90.000,C 0.000} C_DIS
LIN {X -154.635,Y -245.332,Z 103.637,A 57.776,B 90.000,C 0.000} C_DIS
LIN {X -155.509,Y -244.779,Z 101.361,A 57.572,B 90.000,C 0.000} C_DIS
LIN {X -156.420,Y -244.198,Z 99.107,A 57.359,B 90.000,C 0.000} C_DIS
LIN {X -157.489,Y -243.510,Z 96.954,A 57.107,B 90.000,C 0.000} C_DIS
LIN {X -158.609,Y -242.782,Z 94.841,A 56.844,B 90.000,C 0.000} C_DIS
LIN {X -159.817,Y -241.988,Z 92.802,A 56.558,B 90.000,C 0.000} C_DIS
LIN {X -161.011,Y -241.193,Z 90.755,A 56.274,B 90.000,C 0.000} C_DIS
LIN {X -161.990,Y -240.540,Z 89.067,A 56.042,B 90.000,C 0.000} C_DIS
LIN {X -162.978,Y -239.871,Z 86.870,A 55.806,B 90.000,C 0.000} C_DIS
LIN {X -163.927,Y -239.223,Z 84.650,A 55.579,B 90.000,C 0.000} C_DIS
LIN {X -163.993,Y -239.178,Z 84.492,A 55.563,B 90.000,C 0.000} C_DIS
LIN {X -164.980,Y -238.498,Z 86.686,A 55.327,B 90.000,C 0.000} C_DIS
LIN {X -166.101,Y -237.719,Z 88.780,A 55.057,B 90.000,C 0.000} C_DIS
LIN {X -167.427,Y -236.787,Z 90.684,A 54.737,B 90.000,C 0.000} C_DIS
LIN {X -168.796,Y -235.809,Z 92.533,A 54.404,B 90.000,C 0.000} C_DIS
LIN {X -170.156,Y -234.834,Z 94.390,A 54.074,B 90.000,C 0.000} C_DIS
LIN {X -170.327,Y -234.710,Z 94.629,A 54.032,B 90.000,C 0.000} C_DIS
LIN {X -170.737,Y -234.412,Z 94.937,A 53.932,B 90.000,C 0.000} C_DIS
LIN {X -171.210,Y -234.066,Z 95.007,A 53.816,B 90.000,C 0.000} C_DIS
LIN {X -171.468,Y -233.878,Z 94.952,A 53.753,B 90.000,C 0.000} C_DIS
LIN {X -171.651,Y -233.743,Z 94.786,A 53.708,B 90.000,C 0.000} C_DIS
LIN {X -172.709,Y -232.960,Z 92.661,A 53.448,B 90.000,C 0.000} C_DIS
LIN {X -173.724,Y -232.207,Z 90.504,A 53.198,B 90.000,C 0.000} C_DIS
LIN {X -174.839,Y -231.367,Z 88.430,A 52.923,B 90.000,C 0.000} C_DIS
LIN {X -175.152,Y -231.131,Z 87.849,A 52.845,B 90.000,C 0.000} C_DIS
LIN {X -176.487,Y -230.113,Z 85.996,A 52.513,B 90.000,C 0.000} C_DIS
LIN {X -176.749,Y -229.912,Z 85.632,A 52.448,B 90.000,C 0.000} C_DIS
LIN {X -177.279,Y -229.504,Z 85.091,A 52.316,B 90.000,C 0.000} C_DIS
LIN {X -177.941,Y -228.992,Z 84.550,A 52.151,B 90.000,C 0.000} C_DIS
LIN {X -179.710,Y -227.605,Z 83.455,A 51.707,B 90.000,C 0.000} C_DIS
LIN {X -180.551,Y -226.939,Z 82.946,A 51.494,B 90.000,C 0.000} C_DIS
LIN {X -180.847,Y -226.704,Z 82.657,A 51.420,B 90.000,C 0.000} C_DIS
LIN {X -181.015,Y -226.569,Z 82.367,A 51.377,B 90.000,C 0.000} C_DIS
LIN {X -181.106,Y -226.496,Z 81.801,A 51.354,B 90.000,C 0.000} C_DIS
LIN {X -181.037,Y -226.551,Z 81.177,A 51.372,B 90.000,C 0.000} C_DIS
LIN {X -180.787,Y -226.751,Z 80.659,A 51.435,B 90.000,C 0.000} C_DIS
LIN {X -180.429,Y -227.036,Z 80.311,A 51.525,B 90.000,C 0.000} C_DIS
LIN {X -179.808,Y -227.528,Z 80.217,A 51.682,B 90.000,C 0.000} C_DIS
LIN {X -177.864,Y -229.051,Z 80.609,A 52.170,B 90.000,C 0.000} C_DIS
LIN {X -175.889,Y -230.567,Z 80.828,A 52.662,B 90.000,C 0.000} C_DIS
LIN {X -173.898,Y -232.076,Z 80.935,A 53.155,B 90.000,C 0.000} C_DIS
LIN {X -171.892,Y -233.564,Z 81.042,A 53.649,B 90.000,C 0.000} C_DIS
LIN {X -170.696,Y -234.441,Z 81.091,A 53.942,B 90.000,C 0.000} C_DIS
LIN {X -170.730,Y -234.417,Z 80.957,A 53.933,B 90.000,C 0.000} C_DIS
LIN {X -170.971,Y -234.241,Z 80.482,A 53.875,B 90.000,C 0.000} C_DIS
LIN {X -172.498,Y -233.119,Z 78.852,A 53.500,B 90.000,C 0.000} C_DIS
LIN {X -173.112,Y -232.663,Z 78.197,A 53.349,B 90.000,C 0.000} C_DIS
LIN {X -174.966,Y -231.270,Z 77.262,A 52.891,B 90.000,C 0.000} C_DIS
LIN {X -176.879,Y -229.812,Z 76.583,A 52.416,B 90.000,C 0.000} C_DIS
LIN {X -178.840,Y -228.284,Z 76.316,A 51.924,B 90.000,C 0.000} C_DIS
LIN {X -180.802,Y -226.736,Z 76.265,A 51.431,B 90.000,C 0.000} C_DIS
LIN {X -182.749,Y -225.167,Z 76.261,A 50.937,B 90.000,C 0.000} C_DIS
LIN {X -184.684,Y -223.586,Z 76.333,A 50.443,B 90.000,C 0.000} C_DIS
LIN {X -185.517,Y -222.898,Z 76.399,A 50.230,B 90.000,C 0.000} C_DIS
LIN {X -186.860,Y -221.773,Z 76.749,A 49.884,B 90.000,C 0.000} C_DIS
LIN {X -188.663,Y -220.240,Z 77.554,A 49.416,B 90.000,C 0.000} C_DIS
LIN {X -189.625,Y -219.413,Z 78.068,A 49.165,B 90.000,C 0.000} C_DIS
LIN {X -191.108,Y -218.123,Z 79.613,A 48.777,B 90.000,C 0.000} C_DIS
LIN {X -191.675,Y -217.625,Z 80.263,A 48.628,B 90.000,C 0.000} C_DIS
LIN {X -191.954,Y -217.379,Z 80.743,A 48.554,B 90.000,C 0.000} C_DIS
LIN {X -192.027,Y -217.315,Z 80.956,A 48.535,B 90.000,C 0.000} C_DIS
LIN {X -192.006,Y -217.334,Z 81.061,A 48.541,B 90.000,C 0.000} C_DIS
LIN {X -190.124,Y -218.978,Z 81.002,A 49.034,B 90.000,C 0.000} C_DIS
LIN {X -188.229,Y -220.605,Z 80.886,A 49.528,B 90.000,C 0.000} C_DIS
LIN {X -186.327,Y -222.220,Z 80.741,A 50.021,B 90.000,C 0.000} C_DIS
LIN {X -184.423,Y -223.803,Z 80.395,A 50.510,B 90.000,C 0.000} C_DIS
LIN {X -183.329,Y -224.701,Z 80.209,A 50.790,B 90.000,C 0.000} C_DIS
LIN {X -182.702,Y -225.211,Z 80.318,A 50.949,B 90.000,C 0.000} C_DIS
LIN {X -182.446,Y -225.418,Z 80.531,A 51.014,B 90.000,C 0.000} C_DIS
LIN {X -182.248,Y -225.579,Z 80.829,A 51.065,B 90.000,C 0.000} C_DIS
LIN {X -182.118,Y -225.683,Z 81.190,A 51.098,B 90.000,C 0.000} C_DIS
LIN {X -182.069,Y -225.723,Z 81.590,A 51.110,B 90.000,C 0.000} C_DIS
LIN {X -182.137,Y -225.668,Z 82.150,A 51.093,B 90.000,C 0.000} C_DIS
LIN {X -182.385,Y -225.467,Z 82.629,A 51.030,B 90.000,C 0.000} C_DIS
LIN {X -182.841,Y -225.098,Z 83.080,A 50.914,B 90.000,C 0.000} C_DIS
LIN {X -184.598,Y -223.659,Z 84.125,A 50.465,B 90.000,C 0.000} C_DIS
LIN {X -185.274,Y -223.099,Z 84.607,A 50.292,B 90.000,C 0.000} C_DIS
LIN {X -186.755,Y -221.861,Z 86.196,A 49.910,B 90.000,C 0.000} C_DIS
LIN {X -187.482,Y -221.248,Z 87.159,A 49.723,B 90.000,C 0.000} C_DIS
LIN {X -188.598,Y -220.296,Z 89.183,A 49.433,B 90.000,C 0.000} C_DIS
LIN {X -189.651,Y -219.391,Z 91.262,A 49.159,B 90.000,C 0.000} C_DIS
LIN {X -190.567,Y -218.596,Z 93.448,A 48.919,B 90.000,C 0.000} C_DIS
LIN {X -191.074,Y -218.153,Z 94.697,A 48.786,B 90.000,C 0.000} C_DIS
LIN {X -191.278,Y -217.974,Z 94.931,A 48.732,B 90.000,C 0.000} C_DIS
LIN {X -191.540,Y -217.744,Z 95.054,A 48.663,B 90.000,C 0.000} C_DIS
LIN {X -191.828,Y -217.490,Z 95.058,A 48.587,B 90.000,C 0.000} C_DIS
LIN {X -192.113,Y -217.239,Z 94.937,A 48.512,B 90.000,C 0.000} C_DIS
LIN {X -192.576,Y -216.828,Z 94.424,A 48.390,B 90.000,C 0.000} C_DIS
LIN {X -193.792,Y -215.741,Z 92.529,A 48.068,B 90.000,C 0.000} C_DIS
LIN {X -195.036,Y -214.617,Z 90.675,A 47.737,B 90.000,C 0.000} C_DIS
LIN {X -196.254,Y -213.504,Z 88.797,A 47.411,B 90.000,C 0.000} C_DIS
LIN {X -196.879,Y -212.929,Z 87.676,A 47.243,B 90.000,C 0.000} C_DIS
LIN {X -197.765,Y -212.105,Z 85.488,A 47.004,B 90.000,C 0.000} C_DIS
LIN {X -198.174,Y -211.724,Z 84.492,A 46.893,B 90.000,C 0.000} C_DIS
LIN {X -198.957,Y -210.988,Z 86.750,A 46.681,B 90.000,C 0.000} C_DIS
LIN {X -199.880,Y -210.114,Z 88.902,A 46.430,B 90.000,C 0.000} C_DIS
LIN {X -200.885,Y -209.152,Z 90.979,A 46.155,B 90.000,C 0.000} C_DIS
LIN {X -201.912,Y -208.160,Z 93.031,A 45.873,B 90.000,C 0.000} C_DIS
LIN {X -202.935,Y -207.165,Z 95.084,A 45.591,B 90.000,C 0.000} C_DIS
LIN {X -203.893,Y -206.222,Z 97.191,A 45.325,B 90.000,C 0.000} C_DIS
LIN {X -204.763,Y -205.359,Z 99.370,A 45.083,B 90.000,C 0.000} C_DIS
LIN {X -205.515,Y -204.606,Z 101.632,A 44.873,B 90.000,C 0.000} C_DIS
LIN {X -206.316,Y -203.798,Z 103.859,A 44.648,B 90.000,C 0.000} C_DIS
LIN {X -207.262,Y -202.836,Z 105.963,A 44.382,B 90.000,C 0.000} C_DIS
LIN {X -207.806,Y -202.279,Z 107.033,A 44.228,B 90.000,C 0.000} C_DIS
LIN {X -207.872,Y -202.211,Z 107.292,A 44.209,B 90.000,C 0.000} C_DIS
LIN {X -207.265,Y -202.833,Z 106.993,A 44.381,B 90.000,C 0.000} C_DIS
LIN {X -206.342,Y -203.772,Z 106.273,A 44.641,B 90.000,C 0.000} C_DIS
LIN {X -205.563,Y -204.558,Z 105.416,A 44.860,B 90.000,C 0.000} C_DIS
LIN {X -204.366,Y -205.753,Z 103.575,A 45.194,B 90.000,C 0.000} C_DIS
LIN {X -203.271,Y -206.834,Z 101.605,A 45.498,B 90.000,C 0.000} C_DIS
LIN {X -202.207,Y -207.875,Z 99.597,A 45.792,B 90.000,C 0.000} C_DIS
LIN {X -201.132,Y -208.911,Z 97.591,A 46.087,B 90.000,C 0.000} C_DIS
LIN {X -200.057,Y -209.945,Z 95.585,A 46.381,B 90.000,C 0.000} C_DIS
LIN {X -199.026,Y -210.923,Z 93.528,A 46.662,B 90.000,C 0.000} C_DIS
LIN {X -198.381,Y -211.530,Z 92.110,A 46.837,B 90.000,C 0.000} C_DIS
LIN {X -198.154,Y -211.743,Z 91.815,A 46.899,B 90.000,C 0.000} C_DIS
LIN {X -197.906,Y -211.975,Z 91.643,A 46.966,B 90.000,C 0.000} C_DIS
LIN {X -197.665,Y -212.200,Z 91.608,A 47.031,B 90.000,C 0.000} C_DIS
LIN {X -197.459,Y -212.391,Z 91.722,A 47.086,B 90.000,C 0.000} C_DIS
LIN {X -197.237,Y -212.598,Z 92.113,A 47.146,B 90.000,C 0.000} C_DIS
LIN {X -196.435,Y -213.338,Z 94.362,A 47.362,B 90.000,C 0.000} C_DIS
LIN {X -195.866,Y -213.861,Z 95.597,A 47.515,B 90.000,C 0.000} C_DIS
LIN {X -194.720,Y -214.904,Z 97.557,A 47.821,B 90.000,C 0.000} C_DIS
LIN {X -194.075,Y -215.487,Z 98.701,A 47.993,B 90.000,C 0.000} C_DIS
LIN {X -193.540,Y -215.969,Z 100.126,A 48.135,B 90.000,C 0.000} C_DIS
LIN {X -193.394,Y -216.099,Z 100.776,A 48.174,B 90.000,C 0.000} C_DIS
LIN {X -193.110,Y -216.353,Z 103.247,A 48.249,B 90.000,C 0.000} C_DIS
LIN {X -192.864,Y -216.572,Z 104.638,A 48.314,B 90.000,C 0.000} C_DIS
LIN {X -192.055,Y -217.290,Z 106.892,A 48.528,B 90.000,C 0.000} C_DIS
LIN {X -191.866,Y -217.457,Z 107.349,A 48.577,B 90.000,C 0.000} C_DIS
LIN {X -190.488,Y -218.664,Z 109.050,A 48.939,B 90.000,C 0.000} C_DIS
LIN {X -190.306,Y -218.824,Z 109.256,A 48.987,B 90.000,C 0.000} C_DIS
LIN {X -189.511,Y -219.512,Z 109.881,A 49.195,B 90.000,C 0.000} C_DIS
LIN {X -188.227,Y -220.614,Z 110.248,A 49.529,B 90.000,C 0.000} C_DIS
LIN {X -188.100,Y -220.723,Z 110.362,A 49.562,B 90.000,C 0.000} C_DIS
LIN {X -188.048,Y -220.767,Z 110.512,A 49.576,B 90.000,C 0.000} C_DIS
LIN {X -188.135,Y -220.692,Z 111.105,A 49.553,B 90.000,C 0.000} C_DIS
LIN {X -188.377,Y -220.486,Z 111.881,A 49.490,B 90.000,C 0.000} C_DIS
LIN {X -188.714,Y -220.197,Z 112.510,A 49.403,B 90.000,C 0.000} C_DIS
LIN {X -189.103,Y -219.864,Z 112.927,A 49.302,B 90.000,C 0.000} C_DIS
LIN {X -189.589,Y -219.445,Z 113.122,A 49.175,B 90.000,C 0.000} C_DIS
LIN {X -190.193,Y -218.922,Z 113.152,A 49.017,B 90.000,C 0.000} C_DIS
LIN {X -190.878,Y -218.325,Z 113.021,A 48.837,B 90.000,C 0.000} C_DIS
LIN {X -191.608,Y -217.684,Z 112.730,A 48.645,B 90.000,C 0.000} C_DIS
LIN {X -192.361,Y -217.019,Z 112.290,A 48.447,B 90.000,C 0.000} C_DIS
LIN {X -192.996,Y -216.454,Z 111.755,A 48.279,B 90.000,C 0.000} C_DIS
LIN {X -193.583,Y -215.929,Z 111.056,A 48.123,B 90.000,C 0.000} C_DIS
LIN {X -194.748,Y -214.880,Z 109.109,A 47.814,B 90.000,C 0.000} C_DIS
LIN {X -194.841,Y -214.795,Z 108.939,A 47.789,B 90.000,C 0.000} C_DIS
LIN {X -195.752,Y -213.965,Z 106.764,A 47.545,B 90.000,C 0.000} C_DIS
LIN {X -196.605,Y -213.182,Z 104.549,A 47.317,B 90.000,C 0.000} C_DIS
LIN {X -197.288,Y -212.549,Z 102.229,A 47.133,B 90.000,C 0.000} C_DIS
LIN {X -197.941,Y -211.942,Z 99.893,A 46.956,B 90.000,C 0.000} C_DIS
LIN {X -198.148,Y -211.748,Z 99.151,A 46.900,B 90.000,C 0.000} C_DIS
LIN {X -198.224,Y -211.677,Z 99.168,A 46.880,B 90.000,C 0.000} C_DIS
LIN {X -199.125,Y -210.828,Z 101.339,A 46.635,B 90.000,C 0.000} C_DIS
LIN {X -200.038,Y -209.963,Z 103.500,A 46.387,B 90.000,C 0.000} C_DIS
LIN {X -200.881,Y -209.158,Z 105.460,A 46.156,B 90.000,C 0.000} C_DIS
LIN {X -201.414,Y -208.644,Z 106.292,A 46.010,B 90.000,C 0.000} C_DIS
LIN {X -202.092,Y -207.988,Z 106.813,A 45.824,B 90.000,C 0.000} C_DIS
LIN {X -203.797,Y -206.315,Z 107.552,A 45.352,B 90.000,C 0.000} C_DIS
LIN {X -204.319,Y -205.801,Z 107.782,A 45.207,B 90.000,C 0.000} C_DIS
LIN {X -205.204,Y -204.918,Z 108.488,A 44.960,B 90.000,C 0.000} C_DIS
LIN {X -205.544,Y -204.577,Z 108.859,A 44.865,B 90.000,C 0.000} C_DIS
LIN {X -205.806,Y -204.313,Z 109.265,A 44.791,B 90.000,C 0.000} C_DIS
LIN {X -206.009,Y -204.108,Z 109.740,A 44.734,B 90.000,C 0.000} C_DIS
LIN {X -206.171,Y -203.945,Z 110.318,A 44.689,B 90.000,C 0.000} C_DIS
LIN {X -206.243,Y -203.872,Z 110.804,A 44.669,B 90.000,C 0.000} C_DIS
LIN {X -206.069,Y -204.048,Z 111.041,A 44.718,B 90.000,C 0.000} C_DIS
LIN {X -205.554,Y -204.567,Z 111.318,A 44.862,B 90.000,C 0.000} C_DIS
LIN {X -203.805,Y -206.309,Z 111.720,A 45.350,B 90.000,C 0.000} C_DIS
LIN {X -203.734,Y -206.380,Z 111.737,A 45.370,B 90.000,C 0.000} C_DIS
LIN {X -202.985,Y -207.116,Z 112.117,A 45.577,B 90.000,C 0.000} C_DIS
LIN {X -202.119,Y -207.961,Z 112.768,A 45.816,B 90.000,C 0.000} C_DIS
LIN {X -200.648,Y -209.380,Z 114.207,A 46.220,B 90.000,C 0.000} C_DIS
LIN {X -200.134,Y -209.873,Z 114.732,A 46.361,B 90.000,C 0.000} C_DIS
LIN {X -199.560,Y -210.418,Z 117.095,A 46.517,B 90.000,C 0.000} C_DIS
LIN {X -199.484,Y -210.490,Z 117.825,A 46.538,B 90.000,C 0.000} C_DIS
LIN {X -199.477,Y -210.497,Z 118.544,A 46.540,B 90.000,C 0.000} C_DIS
LIN {X -199.607,Y -210.374,Z 119.623,A 46.504,B 90.000,C 0.000} C_DIS
LIN {X -200.321,Y -209.694,Z 121.730,A 46.310,B 90.000,C 0.000} C_DIS
LIN {X -201.965,Y -208.110,Z 122.749,A 45.858,B 90.000,C 0.000} C_DIS
LIN {X -202.225,Y -207.858,Z 122.950,A 45.787,B 90.000,C 0.000} C_DIS
LIN {X -203.586,Y -206.524,Z 124.568,A 45.410,B 90.000,C 0.000} C_DIS
LIN {X -204.070,Y -206.047,Z 125.161,A 45.276,B 90.000,C 0.000} C_DIS
LIN {X -204.598,Y -205.523,Z 125.498,A 45.129,B 90.000,C 0.000} C_DIS
LIN {X -205.213,Y -204.908,Z 125.664,A 44.957,B 90.000,C 0.000} C_DIS
LIN {X -205.865,Y -204.254,Z 125.653,A 44.775,B 90.000,C 0.000} C_DIS
LIN {X -206.500,Y -203.612,Z 125.457,A 44.597,B 90.000,C 0.000} C_DIS
LIN {X -206.905,Y -203.200,Z 125.226,A 44.482,B 90.000,C 0.000} C_DIS
LIN {X -207.166,Y -202.934,Z 124.843,A 44.409,B 90.000,C 0.000} C_DIS
LIN {X -207.339,Y -202.758,Z 124.480,A 44.360,B 90.000,C 0.000} C_DIS
LIN {X -207.400,Y -202.695,Z 124.137,A 44.343,B 90.000,C 0.000} C_DIS
LIN {X -207.350,Y -202.746,Z 123.739,A 44.357,B 90.000,C 0.000} C_DIS
LIN {X -207.039,Y -203.064,Z 122.692,A 44.445,B 90.000,C 0.000} C_DIS
LIN {X -206.969,Y -203.135,Z 122.157,A 44.464,B 90.000,C 0.000} C_DIS
LIN {X -206.962,Y -203.143,Z 119.657,A 44.466,B 90.000,C 0.000} C_DIS
LIN {X -207.014,Y -203.089,Z 117.861,A 44.452,B 90.000,C 0.000} C_DIS
LIN {X -207.349,Y -202.747,Z 115.408,A 44.357,B 90.000,C 0.000} C_DIS
LIN {X -207.500,Y -202.592,Z 114.655,A 44.314,B 90.000,C 0.000} C_DIS
LIN {X -207.692,Y -202.396,Z 113.995,A 44.260,B 90.000,C 0.000} C_DIS
LIN {X -208.050,Y -202.028,Z 113.326,A 44.159,B 90.000,C 0.000} C_DIS
LIN {X -208.413,Y -201.653,Z 112.835,A 44.056,B 90.000,C 0.000} C_DIS
LIN {X -208.896,Y -201.152,Z 112.557,A 43.918,B 90.000,C 0.000} C_DIS
LIN {X -209.488,Y -200.537,Z 112.458,A 43.749,B 90.000,C 0.000} C_DIS
LIN {X -209.848,Y -200.160,Z 112.481,A 43.646,B 90.000,C 0.000} C_DIS
LIN {X -210.064,Y -199.933,Z 112.612,A 43.584,B 90.000,C 0.000} C_DIS
LIN {X -210.248,Y -199.740,Z 112.826,A 43.532,B 90.000,C 0.000} C_DIS
LIN {X -210.408,Y -199.571,Z 113.151,A 43.486,B 90.000,C 0.000} C_DIS
LIN {X -210.722,Y -199.239,Z 114.305,A 43.396,B 90.000,C 0.000} C_DIS
LIN {X -211.167,Y -198.767,Z 116.720,A 43.267,B 90.000,C 0.000} C_DIS
LIN {X -211.557,Y -198.352,Z 119.154,A 43.155,B 90.000,C 0.000} C_DIS
LIN {X -211.816,Y -198.075,Z 120.930,A 43.080,B 90.000,C 0.000} C_DIS
LIN {X -211.958,Y -197.923,Z 123.352,A 43.039,B 90.000,C 0.000} C_DIS
LIN {X -211.908,Y -197.978,Z 125.670,A 43.054,B 90.000,C 0.000} C_DIS
LIN {X -211.595,Y -198.311,Z 128.128,A 43.144,B 90.000,C 0.000} C_DIS
LIN {X -211.137,Y -198.800,Z 130.537,A 43.276,B 90.000,C 0.000} C_DIS
LIN {X -210.678,Y -199.285,Z 132.946,A 43.408,B 90.000,C 0.000} C_DIS
LIN {X -210.250,Y -199.737,Z 135.367,A 43.531,B 90.000,C 0.000} C_DIS
LIN {X -209.918,Y -200.086,Z 137.820,A 43.626,B 90.000,C 0.000} C_DIS
LIN {X -209.724,Y -200.289,Z 140.304,A 43.682,B 90.000,C 0.000} C_DIS
LIN {X -209.687,Y -200.329,Z 141.174,A 43.693,B 90.000,C 0.000} C_DIS
LIN {X -209.758,Y -200.254,Z 142.717,A 43.672,B 90.000,C 0.000} C_DIS
LIN {X -210.038,Y -199.960,Z 144.375,A 43.592,B 90.000,C 0.000} C_DIS
LIN {X -210.750,Y -199.209,Z 146.651,A 43.387,B 90.000,C 0.000} C_DIS
LIN {X -211.473,Y -198.441,Z 148.917,A 43.179,B 90.000,C 0.000} C_DIS
LIN {X -212.186,Y -197.677,Z 151.188,A 42.973,B 90.000,C 0.000} C_DIS
LIN {X -212.887,Y -196.924,Z 153.467,A 42.769,B 90.000,C 0.000} C_DIS
LIN {X -213.164,Y -196.624,Z 154.389,A 42.689,B 90.000,C 0.000} C_DIS
LIN {X -213.585,Y -196.167,Z 156.811,A 42.566,B 90.000,C 0.000} C_DIS
LIN {X -213.950,Y -195.769,Z 159.251,A 42.459,B 90.000,C 0.000} C_DIS
LIN {X -214.208,Y -195.486,Z 161.722,A 42.384,B 90.000,C 0.000} C_DIS
LIN {X -214.356,Y -195.325,Z 164.212,A 42.340,B 90.000,C 0.000} C_DIS
LIN {X -214.393,Y -195.284,Z 166.712,A 42.329,B 90.000,C 0.000} C_DIS
LIN {X -214.380,Y -195.298,Z 169.211,A 42.333,B 90.000,C 0.000} C_DIS
LIN {X -214.372,Y -195.306,Z 170.270,A 42.335,B 90.000,C 0.000} C_DIS
LIN {X -214.459,Y -195.212,Z 171.592,A 42.310,B 90.000,C 0.000} C_DIS
LIN {X -214.646,Y -195.005,Z 172.071,A 42.255,B 90.000,C 0.000} C_DIS
LIN {X -214.920,Y -194.703,Z 172.225,A 42.174,B 90.000,C 0.000} C_DIS
LIN {X -215.198,Y -194.396,Z 172.105,A 42.093,B 90.000,C 0.000} C_DIS
LIN {X -215.394,Y -194.179,Z 171.610,A 42.035,B 90.000,C 0.000} C_DIS
LIN {X -215.955,Y -193.554,Z 169.594,A 41.869,B 90.000,C 0.000} C_DIS
LIN {X -216.115,Y -193.376,Z 168.559,A 41.822,B 90.000,C 0.000} C_DIS
LIN {X -216.302,Y -193.167,Z 166.075,A 41.766,B 90.000,C 0.000} C_DIS
LIN {X -216.433,Y -193.020,Z 163.583,A 41.727,B 90.000,C 0.000} C_DIS
LIN {X -216.542,Y -192.897,Z 161.088,A 41.695,B 90.000,C 0.000} C_DIS
LIN {X -216.587,Y -192.848,Z 158.589,A 41.682,B 90.000,C 0.000} C_DIS
LIN {X -216.603,Y -192.830,Z 156.107,A 41.677,B 90.000,C 0.000} C_DIS
LIN {X -216.458,Y -192.992,Z 153.616,A 41.720,B 90.000,C 0.000} C_DIS
LIN {X -216.361,Y -193.101,Z 151.120,A 41.749,B 90.000,C 0.000} C_DIS
LIN {X -216.254,Y -193.221,Z 148.626,A 41.781,B 90.000,C 0.000} C_DIS
LIN {X -216.207,Y -193.274,Z 148.142,A 41.795,B 90.000,C 0.000} C_DIS
LIN {X -216.084,Y -193.411,Z 147.580,A 41.831,B 90.000,C 0.000} C_DIS
LIN {X -215.930,Y -193.583,Z 147.190,A 41.876,B 90.000,C 0.000} C_DIS
LIN {X -215.727,Y -193.809,Z 146.908,A 41.936,B 90.000,C 0.000} C_DIS
LIN {X -215.478,Y -194.085,Z 146.737,A 42.010,B 90.000,C 0.000} C_DIS
LIN {X -215.186,Y -194.409,Z 146.680,A 42.096,B 90.000,C 0.000} C_DIS
LIN {X -214.758,Y -194.882,Z 146.856,A 42.222,B 90.000,C 0.000} C_DIS
LIN {X -213.897,Y -195.826,Z 147.911,A 42.475,B 90.000,C 0.000} C_DIS
LIN {X -213.783,Y -195.951,Z 147.979,A 42.508,B 90.000,C 0.000} C_DIS
LIN {X -213.407,Y -196.361,Z 145.542,A 42.618,B 90.000,C 0.000} C_DIS
LIN {X -213.151,Y -196.638,Z 143.071,A 42.692,B 90.000,C 0.000} C_DIS
LIN {X -213.068,Y -196.728,Z 140.574,A 42.717,B 90.000,C 0.000} C_DIS
LIN {X -213.098,Y -196.696,Z 138.074,A 42.708,B 90.000,C 0.000} C_DIS
LIN {X -213.106,Y -196.687,Z 137.489,A 42.706,B 90.000,C 0.000} C_DIS
LIN {X -213.348,Y -196.425,Z 135.129,A 42.635,B 90.000,C 0.000} C_DIS
LIN {X -213.743,Y -195.994,Z 133.235,A 42.520,B 90.000,C 0.000} C_DIS
LIN {X -214.678,Y -194.969,Z 135.314,A 42.245,B 90.000,C 0.000} C_DIS
LIN {X -215.660,Y -193.883,Z 137.341,A 41.956,B 90.000,C 0.000} C_DIS
LIN {X -215.828,Y -193.696,Z 137.660,A 41.907,B 90.000,C 0.000} C_DIS
LIN {X -216.507,Y -192.937,Z 138.645,A 41.705,B 90.000,C 0.000} C_DIS
LIN {X -217.226,Y -192.127,Z 139.386,A 41.491,B 90.000,C 0.000} C_DIS
LIN {X -217.852,Y -191.417,Z 139.834,A 41.304,B 90.000,C 0.000} C_DIS
LIN {X -218.400,Y -190.791,Z 140.052,A 41.140,B 90.000,C 0.000} C_DIS
LIN {X -218.820,Y -190.310,Z 140.030,A 41.014,B 90.000,C 0.000} C_DIS
LIN {X -218.966,Y -190.142,Z 139.925,A 40.970,B 90.000,C 0.000} C_DIS
LIN {X -219.060,Y -190.033,Z 139.757,A 40.941,B 90.000,C 0.000} C_DIS
LIN {X -219.608,Y -189.399,Z 137.401,A 40.776,B 90.000,C 0.000} C_DIS
LIN {X -220.185,Y -188.728,Z 135.221,A 40.601,B 90.000,C 0.000} C_DIS
LIN {X -220.301,Y -188.593,Z 134.156,A 40.566,B 90.000,C 0.000} C_DIS
RET=EKI_SetBool("oxy","torchState",FALSE)
RET = EKI_Send("oxy","torchState")
PTP {X -218.782,Y -187.293,Z 134.156,A 40.566,B 90.000,C 0.000}
PTP {X -205.108,Y -175.587,Z 134.156,A 40.566,B 90.000,C 0.000}
PTP {X -202.932,Y -178.097,Z 141.106,A 41.271,B 90.000,C 0.000}
PTP {X -216.461,Y -189.970,Z 141.106,A 41.271,B 90.000,C 0.000}
WAIT SEC 2
RET=EKI_SetBool("oxy","torchState",TRUE)
RET = EKI_Send("oxy","torchState")
LIN {X -217.964,Y -191.289,Z 141.106,A 41.271,B 90.000,C 0.000} C_DIS
LIN {X -219.415,Y -189.624,Z 142.057,A 40.834,B 90.000,C 0.000} C_DIS
LIN {X -219.872,Y -189.093,Z 142.511,A 40.696,B 90.000,C 0.000} C_DIS
LIN {X -220.244,Y -188.660,Z 143.026,A 40.583,B 90.000,C 0.000} C_DIS
LIN {X -220.581,Y -188.265,Z 143.700,A 40.481,B 90.000,C 0.000} C_DIS
LIN {X -220.835,Y -187.968,Z 144.625,A 40.403,B 90.000,C 0.000} C_DIS
LIN {X -221.012,Y -187.760,Z 145.644,A 40.349,B 90.000,C 0.000} C_DIS
LIN {X -221.158,Y -187.587,Z 147.831,A 40.305,B 90.000,C 0.000} C_DIS
LIN {X -221.112,Y -187.642,Z 148.754,A 40.319,B 90.000,C 0.000} C_DIS
LIN {X -220.995,Y -187.780,Z 149.394,A 40.355,B 90.000,C 0.000} C_DIS
LIN {X -220.810,Y -187.997,Z 149.976,A 40.411,B 90.000,C 0.000} C_DIS
LIN {X -220.591,Y -188.254,Z 150.418,A 40.478,B 90.000,C 0.000} C_DIS
LIN {X -220.368,Y -188.515,Z 150.638,A 40.545,B 90.000,C 0.000} C_DIS
LIN {X -220.251,Y -188.652,Z 150.623,A 40.581,B 90.000,C 0.000} C_DIS
LIN {X -220.103,Y -188.824,Z 150.490,A 40.626,B 90.000,C 0.000} C_DIS
LIN {X -219.037,Y -190.060,Z 148.782,A 40.948,B 90.000,C 0.000} C_DIS
LIN {X -217.696,Y -191.594,Z 147.334,A 41.351,B 90.000,C 0.000} C_DIS
LIN {X -216.243,Y -193.232,Z 146.127,A 41.784,B 90.000,C 0.000} C_DIS
LIN {X -215.932,Y -193.580,Z 145.876,A 41.876,B 90.000,C 0.000} C_DIS
LIN {X -214.913,Y -194.711,Z 144.729,A 42.177,B 90.000,C 0.000} C_DIS
LIN {X -214.600,Y -195.056,Z 144.223,A 42.269,B 90.000,C 0.000} C_DIS
LIN {X -214.377,Y -195.301,Z 143.705,A 42.334,B 90.000,C 0.000} C_DIS
LIN {X -214.233,Y -195.459,Z 143.149,A 42.376,B 90.000,C 0.000} C_DIS
LIN {X -214.149,Y -195.551,Z 142.441,A 42.401,B 90.000,C 0.000} C_DIS
LIN {X -214.083,Y -195.623,Z 139.943,A 42.420,B 90.000,C 0.000} C_DIS
LIN {X -214.139,Y -195.562,Z 137.920,A 42.404,B 90.000,C 0.000} C_DIS
LIN {X -214.284,Y -195.404,Z 137.232,A 42.361,B 90.000,C 0.000} C_DIS
LIN {X -214.387,Y -195.290,Z 137.063,A 42.331,B 90.000,C 0.000} C_DIS
LIN {X -214.511,Y -195.154,Z 137.007,A 42.295,B 90.000,C 0.000} C_DIS
LIN {X -214.840,Y -194.792,Z 137.367,A 42.198,B 90.000,C 0.000} C_DIS
LIN {X -215.652,Y -193.893,Z 139.159,A 41.959,B 90.000,C 0.000} C_DIS
LIN {X -216.160,Y -193.326,Z 139.837,A 41.808,B 90.000,C 0.000} C_DIS
LIN {X -216.899,Y -192.496,Z 140.453,A 41.589,B 90.000,C 0.000} C_DIS
LIN {X -217.964,Y -191.289,Z 141.106,A 41.271,B 90.000,C 0.000} C_DIS
RET=EKI_SetBool("oxy","torchState",FALSE)
RET = EKI_Send("oxy","torchState")
PTP {X -216.461,Y -189.970,Z 141.106,A 41.271,B 90.000,C 0.000}
PTP {X -202.932,Y -178.097,Z 141.106,A 41.271,B 90.000,C 0.000}
PTP {X -194.764,Y -186.995,Z 134.012,A 43.834,B 90.000,C 0.000}
PTP {X -207.748,Y -199.461,Z 134.012,A 43.834,B 90.000,C 0.000}
WAIT SEC 2
RET=EKI_SetBool("oxy","torchState",TRUE)
RET = EKI_Send("oxy","torchState")
LIN {X -209.190,Y -200.847,Z 134.012,A 43.834,B 90.000,C 0.000} C_DIS
LIN {X -208.672,Y -201.385,Z 135.131,A 43.982,B 90.000,C 0.000} C_DIS
LIN {X -208.011,Y -202.068,Z 136.230,A 44.170,B 90.000,C 0.000} C_DIS
LIN {X -207.420,Y -202.674,Z 136.981,A 44.337,B 90.000,C 0.000} C_DIS
LIN {X -206.004,Y -204.113,Z 138.456,A 44.736,B 90.000,C 0.000} C_DIS
LIN {X -205.653,Y -204.468,Z 138.838,A 44.834,B 90.000,C 0.000} C_DIS
LIN {X -205.104,Y -205.018,Z 139.738,A 44.988,B 90.000,C 0.000} C_DIS
LIN {X -204.740,Y -205.381,Z 140.586,A 45.090,B 90.000,C 0.000} C_DIS
LIN {X -204.263,Y -205.856,Z 142.188,A 45.223,B 90.000,C 0.000} C_DIS
LIN {X -204.127,Y -205.990,Z 142.378,A 45.260,B 90.000,C 0.000} C_DIS
LIN {X -203.943,Y -206.173,Z 142.507,A 45.312,B 90.000,C 0.000} C_DIS
LIN {X -203.654,Y -206.458,Z 142.573,A 45.392,B 90.000,C 0.000} C_DIS
LIN {X -203.294,Y -206.813,Z 142.494,A 45.492,B 90.000,C 0.000} C_DIS
LIN {X -201.687,Y -208.380,Z 141.394,A 45.935,B 90.000,C 0.000} C_DIS
LIN {X -201.433,Y -208.626,Z 141.202,A 46.005,B 90.000,C 0.000} C_DIS
LIN {X -200.908,Y -209.131,Z 140.946,A 46.149,B 90.000,C 0.000} C_DIS
LIN {X -200.724,Y -209.308,Z 140.949,A 46.199,B 90.000,C 0.000} C_DIS
LIN {X -200.602,Y -209.425,Z 141.066,A 46.233,B 90.000,C 0.000} C_DIS
LIN {X -200.515,Y -209.508,Z 141.246,A 46.256,B 90.000,C 0.000} C_DIS
LIN {X -200.496,Y -209.527,Z 141.543,A 46.262,B 90.000,C 0.000} C_DIS
LIN {X -200.581,Y -209.445,Z 142.285,A 46.238,B 90.000,C 0.000} C_DIS
LIN {X -200.810,Y -209.226,Z 143.137,A 46.176,B 90.000,C 0.000} C_DIS
LIN {X -201.318,Y -208.737,Z 144.072,A 46.037,B 90.000,C 0.000} C_DIS
LIN {X -202.134,Y -207.947,Z 145.005,A 45.812,B 90.000,C 0.000} C_DIS
LIN {X -202.821,Y -207.277,Z 145.542,A 45.623,B 90.000,C 0.000} C_DIS
LIN {X -203.449,Y -206.661,Z 145.775,A 45.449,B 90.000,C 0.000} C_DIS
LIN {X -203.982,Y -206.134,Z 145.796,A 45.301,B 90.000,C 0.000} C_DIS
LIN {X -205.739,Y -204.380,Z 145.507,A 44.810,B 90.000,C 0.000} C_DIS
LIN {X -205.781,Y -204.339,Z 145.500,A 44.799,B 90.000,C 0.000} C_DIS
LIN {X -206.385,Y -203.728,Z 145.529,A 44.629,B 90.000,C 0.000} C_DIS
LIN {X -206.841,Y -203.266,Z 145.717,A 44.501,B 90.000,C 0.000} C_DIS
LIN {X -207.204,Y -202.895,Z 146.077,A 44.398,B 90.000,C 0.000} C_DIS
LIN {X -207.434,Y -202.661,Z 146.477,A 44.333,B 90.000,C 0.000} C_DIS
LIN {X -207.587,Y -202.503,Z 146.969,A 44.290,B 90.000,C 0.000} C_DIS
LIN {X -207.668,Y -202.420,Z 147.564,A 44.267,B 90.000,C 0.000} C_DIS
LIN {X -207.678,Y -202.410,Z 148.273,A 44.264,B 90.000,C 0.000} C_DIS
LIN {X -207.603,Y -202.487,Z 149.036,A 44.285,B 90.000,C 0.000} C_DIS
LIN {X -207.366,Y -202.730,Z 149.554,A 44.352,B 90.000,C 0.000} C_DIS
LIN {X -206.989,Y -203.114,Z 149.956,A 44.459,B 90.000,C 0.000} C_DIS
LIN {X -206.474,Y -203.638,Z 150.223,A 44.604,B 90.000,C 0.000} C_DIS
LIN {X -205.841,Y -204.278,Z 150.348,A 44.782,B 90.000,C 0.000} C_DIS
LIN {X -205.109,Y -205.013,Z 150.323,A 44.986,B 90.000,C 0.000} C_DIS
LIN {X -204.379,Y -205.741,Z 150.177,A 45.190,B 90.000,C 0.000} C_DIS
LIN {X -203.719,Y -206.394,Z 149.935,A 45.374,B 90.000,C 0.000} C_DIS
LIN {X -203.120,Y -206.983,Z 149.586,A 45.540,B 90.000,C 0.000} C_DIS
LIN {X -202.572,Y -207.520,Z 149.120,A 45.691,B 90.000,C 0.000} C_DIS
LIN {X -202.063,Y -208.016,Z 148.524,A 45.832,B 90.000,C 0.000} C_DIS
LIN {X -201.583,Y -208.481,Z 147.788,A 45.964,B 90.000,C 0.000} C_DIS
LIN {X -200.610,Y -209.417,Z 145.685,A 46.231,B 90.000,C 0.000} C_DIS
LIN {X -199.817,Y -210.172,Z 143.437,A 46.447,B 90.000,C 0.000} C_DIS
LIN {X -199.134,Y -210.822,Z 141.502,A 46.633,B 90.000,C 0.000} C_DIS
LIN {X -198.705,Y -211.226,Z 139.611,A 46.749,B 90.000,C 0.000} C_DIS
LIN {X -198.485,Y -211.432,Z 139.148,A 46.809,B 90.000,C 0.000} C_DIS
LIN {X -196.995,Y -212.821,Z 137.700,A 47.211,B 90.000,C 0.000} C_DIS
LIN {X -195.430,Y -214.258,Z 136.382,A 47.631,B 90.000,C 0.000} C_DIS
LIN {X -193.805,Y -215.729,Z 135.180,A 48.064,B 90.000,C 0.000} C_DIS
LIN {X -192.925,Y -216.517,Z 134.557,A 48.298,B 90.000,C 0.000} C_DIS
LIN {X -192.504,Y -216.892,Z 134.517,A 48.409,B 90.000,C 0.000} C_DIS
LIN {X -192.121,Y -217.231,Z 134.614,A 48.510,B 90.000,C 0.000} C_DIS
LIN {X -191.797,Y -217.518,Z 134.853,A 48.596,B 90.000,C 0.000} C_DIS
LIN {X -191.485,Y -217.792,Z 135.283,A 48.678,B 90.000,C 0.000} C_DIS
LIN {X -190.380,Y -218.759,Z 137.306,A 48.968,B 90.000,C 0.000} C_DIS
LIN {X -190.056,Y -219.040,Z 137.870,A 49.053,B 90.000,C 0.000} C_DIS
LIN {X -189.953,Y -219.130,Z 138.411,A 49.080,B 90.000,C 0.000} C_DIS
LIN {X -190.083,Y -219.017,Z 138.826,A 49.046,B 90.000,C 0.000} C_DIS
LIN {X -190.403,Y -218.739,Z 139.380,A 48.962,B 90.000,C 0.000} C_DIS
LIN {X -191.754,Y -217.555,Z 141.119,A 48.607,B 90.000,C 0.000} C_DIS
LIN {X -193.126,Y -216.338,Z 142.819,A 48.245,B 90.000,C 0.000} C_DIS
LIN {X -194.453,Y -215.135,Z 144.561,A 47.891,B 90.000,C 0.000} C_DIS
LIN {X -195.779,Y -213.932,Z 146.306,A 47.537,B 90.000,C 0.000} C_DIS
LIN {X -196.607,Y -213.180,Z 147.397,A 47.316,B 90.000,C 0.000} C_DIS
LIN {X -196.766,Y -213.033,Z 147.802,A 47.273,B 90.000,C 0.000} C_DIS
LIN {X -196.868,Y -212.939,Z 148.360,A 47.246,B 90.000,C 0.000} C_DIS
LIN {X -196.991,Y -212.825,Z 150.854,A 47.213,B 90.000,C 0.000} C_DIS
LIN {X -197.131,Y -212.696,Z 153.308,A 47.175,B 90.000,C 0.000} C_DIS
LIN {X -197.285,Y -212.553,Z 154.308,A 47.133,B 90.000,C 0.000} C_DIS
LIN {X -197.751,Y -212.119,Z 156.095,A 47.008,B 90.000,C 0.000} C_DIS
LIN {X -197.818,Y -212.056,Z 156.658,A 46.989,B 90.000,C 0.000} C_DIS
LIN {X -197.721,Y -212.147,Z 157.332,A 47.016,B 90.000,C 0.000} C_DIS
LIN {X -197.421,Y -212.427,Z 157.999,A 47.097,B 90.000,C 0.000} C_DIS
LIN {X -196.930,Y -212.882,Z 158.636,A 47.229,B 90.000,C 0.000} C_DIS
LIN {X -195.802,Y -213.920,Z 159.617,A 47.532,B 90.000,C 0.000} C_DIS
LIN {X -195.529,Y -214.169,Z 160.026,A 47.605,B 90.000,C 0.000} C_DIS
LIN {X -195.429,Y -214.261,Z 160.488,A 47.632,B 90.000,C 0.000} C_DIS
LIN {X -195.481,Y -214.213,Z 161.046,A 47.618,B 90.000,C 0.000} C_DIS
LIN {X -195.614,Y -214.092,Z 161.541,A 47.582,B 90.000,C 0.000} C_DIS
LIN {X -195.807,Y -213.915,Z 161.937,A 47.531,B 90.000,C 0.000} C_DIS
LIN {X -196.080,Y -213.665,Z 162.265,A 47.457,B 90.000,C 0.000} C_DIS
LIN {X -196.451,Y -213.323,Z 162.556,A 47.358,B 90.000,C 0.000} C_DIS
LIN {X -197.102,Y -212.722,Z 162.876,A 47.183,B 90.000,C 0.000} C_DIS
LIN {X -197.808,Y -212.066,Z 162.974,A 46.992,B 90.000,C 0.000} C_DIS
LIN {X -198.362,Y -211.547,Z 162.894,A 46.842,B 90.000,C 0.000} C_DIS
LIN {X -198.873,Y -211.068,Z 162.507,A 46.704,B 90.000,C 0.000} C_DIS
LIN {X -199.261,Y -210.702,Z 162.074,A 46.599,B 90.000,C 0.000} C_DIS
LIN {X -199.620,Y -210.362,Z 161.493,A 46.501,B 90.000,C 0.000} C_DIS
LIN {X -200.532,Y -209.492,Z 159.334,A 46.252,B 90.000,C 0.000} C_DIS
LIN {X -201.445,Y -208.614,Z 157.179,A 46.002,B 90.000,C 0.000} C_DIS
LIN {X -201.651,Y -208.415,Z 156.739,A 45.945,B 90.000,C 0.000} C_DIS
LIN {X -202.002,Y -208.075,Z 156.370,A 45.848,B 90.000,C 0.000} C_DIS
LIN {X -202.257,Y -207.827,Z 156.240,A 45.778,B 90.000,C 0.000} C_DIS
LIN {X -202.602,Y -207.491,Z 156.220,A 45.683,B 90.000,C 0.000} C_DIS
LIN {X -202.955,Y -207.146,Z 156.258,A 45.586,B 90.000,C 0.000} C_DIS
LIN {X -203.316,Y -206.792,Z 156.394,A 45.486,B 90.000,C 0.000} C_DIS
LIN {X -204.913,Y -205.204,Z 157.479,A 45.041,B 90.000,C 0.000} C_DIS
LIN {X -206.486,Y -203.621,Z 158.606,A 44.600,B 90.000,C 0.000} C_DIS
LIN {X -208.033,Y -202.041,Z 159.773,A 44.163,B 90.000,C 0.000} C_DIS
LIN {X -208.695,Y -201.361,Z 160.284,A 43.975,B 90.000,C 0.000} C_DIS
LIN {X -208.955,Y -201.091,Z 160.747,A 43.901,B 90.000,C 0.000} C_DIS
LIN {X -209.099,Y -200.942,Z 161.331,A 43.860,B 90.000,C 0.000} C_DIS
LIN {X -209.126,Y -200.914,Z 162.045,A 43.853,B 90.000,C 0.000} C_DIS
LIN {X -209.038,Y -201.005,Z 162.897,A 43.878,B 90.000,C 0.000} C_DIS
LIN {X -208.524,Y -201.538,Z 165.285,A 44.024,B 90.000,C 0.000} C_DIS
LIN {X -208.107,Y -201.969,Z 167.712,A 44.143,B 90.000,C 0.000} C_DIS
LIN {X -208.099,Y -201.977,Z 167.759,A 44.145,B 90.000,C 0.000} C_DIS
LIN {X -208.024,Y -202.055,Z 169.511,A 44.166,B 90.000,C 0.000} C_DIS
LIN {X -208.094,Y -201.982,Z 171.034,A 44.146,B 90.000,C 0.000} C_DIS
LIN {X -208.231,Y -201.841,Z 171.666,A 44.107,B 90.000,C 0.000} C_DIS
LIN {X -208.419,Y -201.647,Z 172.231,A 44.054,B 90.000,C 0.000} C_DIS
LIN {X -209.468,Y -200.556,Z 174.221,A 43.755,B 90.000,C 0.000} C_DIS
LIN {X -209.670,Y -200.346,Z 174.597,A 43.697,B 90.000,C 0.000} C_DIS
LIN {X -210.022,Y -199.977,Z 175.674,A 43.597,B 90.000,C 0.000} C_DIS
LIN {X -210.182,Y -199.809,Z 176.955,A 43.551,B 90.000,C 0.000} C_DIS
LIN {X -210.157,Y -199.835,Z 179.454,A 43.558,B 90.000,C 0.000} C_DIS
LIN {X -210.073,Y -199.923,Z 180.889,A 43.582,B 90.000,C 0.000} C_DIS
LIN {X -209.524,Y -200.498,Z 183.259,A 43.739,B 90.000,C 0.000} C_DIS
LIN {X -208.948,Y -201.099,Z 184.810,A 43.903,B 90.000,C 0.000} C_DIS
LIN {X -207.907,Y -202.174,Z 186.813,A 44.199,B 90.000,C 0.000} C_DIS
LIN {X -206.779,Y -203.327,Z 188.723,A 44.518,B 90.000,C 0.000} C_DIS
LIN {X -206.393,Y -203.720,Z 189.288,A 44.626,B 90.000,C 0.000} C_DIS
LIN {X -206.003,Y -204.114,Z 189.661,A 44.736,B 90.000,C 0.000} C_DIS
LIN {X -205.601,Y -204.520,Z 189.922,A 44.849,B 90.000,C 0.000} C_DIS
LIN {X -205.146,Y -204.975,Z 190.028,A 44.976,B 90.000,C 0.000} C_DIS
LIN {X -204.877,Y -205.244,Z 189.846,A 45.051,B 90.000,C 0.000} C_DIS
LIN {X -204.822,Y -205.300,Z 189.426,A 45.067,B 90.000,C 0.000} C_DIS
LIN {X -205.354,Y -204.768,Z 187.883,A 44.918,B 90.000,C 0.000} C_DIS
LIN {X -205.607,Y -204.513,Z 186.779,A 44.847,B 90.000,C 0.000} C_DIS
LIN {X -205.770,Y -204.350,Z 185.499,A 44.802,B 90.000,C 0.000} C_DIS
LIN {X -205.829,Y -204.290,Z 183.000,A 44.785,B 90.000,C 0.000} C_DIS
LIN {X -205.822,Y -204.297,Z 182.489,A 44.787,B 90.000,C 0.000} C_DIS
LIN {X -205.650,Y -204.470,Z 181.352,A 44.835,B 90.000,C 0.000} C_DIS
LIN {X -205.413,Y -204.708,Z 180.588,A 44.902,B 90.000,C 0.000} C_DIS
LIN {X -205.079,Y -205.043,Z 180.001,A 44.995,B 90.000,C 0.000} C_DIS
LIN {X -204.631,Y -205.490,Z 179.571,A 45.120,B 90.000,C 0.000} C_DIS
LIN {X -204.051,Y -206.066,Z 179.276,A 45.282,B 90.000,C 0.000} C_DIS
LIN {X -203.342,Y -206.766,Z 179.163,A 45.478,B 90.000,C 0.000} C_DIS
LIN {X -202.657,Y -207.437,Z 179.254,A 45.668,B 90.000,C 0.000} C_DIS
LIN {X -202.088,Y -207.991,Z 179.587,A 45.825,B 90.000,C 0.000} C_DIS
LIN {X -201.515,Y -208.546,Z 180.247,A 45.982,B 90.000,C 0.000} C_DIS
LIN {X -201.062,Y -208.984,Z 180.949,A 46.107,B 90.000,C 0.000} C_DIS
LIN {X -200.685,Y -209.346,Z 181.762,A 46.210,B 90.000,C 0.000} C_DIS
LIN {X -199.981,Y -210.018,Z 184.064,A 46.402,B 90.000,C 0.000} C_DIS
LIN {X -199.375,Y -210.593,Z 186.204,A 46.567,B 90.000,C 0.000} C_DIS
LIN {X -198.927,Y -211.017,Z 187.391,A 46.689,B 90.000,C 0.000} C_DIS
LIN {X -197.870,Y -212.008,Z 189.428,A 46.976,B 90.000,C 0.000} C_DIS
LIN {X -196.717,Y -213.079,Z 191.371,A 47.286,B 90.000,C 0.000} C_DIS
LIN {X -196.056,Y -213.687,Z 192.505,A 47.464,B 90.000,C 0.000} C_DIS
LIN {X -195.632,Y -214.075,Z 193.523,A 47.578,B 90.000,C 0.000} C_DIS
LIN {X -195.433,Y -214.257,Z 194.325,A 47.631,B 90.000,C 0.000} C_DIS
LIN {X -195.440,Y -214.251,Z 194.597,A 47.629,B 90.000,C 0.000} C_DIS
LIN {X -195.531,Y -214.168,Z 194.759,A 47.605,B 90.000,C 0.000} C_DIS
LIN {X -196.784,Y -213.017,Z 195.006,A 47.268,B 90.000,C 0.000} C_DIS
LIN {X -197.366,Y -212.477,Z 195.242,A 47.112,B 90.000,C 0.000} C_DIS
LIN {X -197.876,Y -212.003,Z 195.595,A 46.974,B 90.000,C 0.000} C_DIS
LIN {X -198.305,Y -211.601,Z 196.064,A 46.858,B 90.000,C 0.000} C_DIS
LIN {X -198.637,Y -211.289,Z 196.649,A 46.768,B 90.000,C 0.000} C_DIS
LIN {X -198.703,Y -211.228,Z 197.129,A 46.750,B 90.000,C 0.000} C_DIS
LIN {X -198.300,Y -211.606,Z 197.781,A 46.859,B 90.000,C 0.000} C_DIS
LIN {X -196.819,Y -212.981,Z 199.252,A 47.258,B 90.000,C 0.000} C_DIS
LIN {X -195.262,Y -214.409,Z 200.589,A 47.676,B 90.000,C 0.000} C_DIS
LIN {X -193.666,Y -215.851,Z 201.862,A 48.101,B 90.000,C 0.000} C_DIS
LIN {X -192.038,Y -217.303,Z 203.084,A 48.532,B 90.000,C 0.000} C_DIS
LIN {X -190.344,Y -218.790,Z 204.164,A 48.977,B 90.000,C 0.000} C_DIS
LIN {X -188.551,Y -220.336,Z 204.967,A 49.445,B 90.000,C 0.000} C_DIS
LIN {X -187.986,Y -220.820,Z 205.168,A 49.592,B 90.000,C 0.000} C_DIS
LIN {X -187.449,Y -221.275,Z 205.212,A 49.731,B 90.000,C 0.000} C_DIS
LIN {X -187.033,Y -221.627,Z 204.835,A 49.839,B 90.000,C 0.000} C_DIS
LIN {X -186.782,Y -221.839,Z 204.514,A 49.904,B 90.000,C 0.000} C_DIS
LIN {X -186.864,Y -221.770,Z 204.287,A 49.882,B 90.000,C 0.000} C_DIS
LIN {X -188.022,Y -220.789,Z 202.300,A 49.583,B 90.000,C 0.000} C_DIS
LIN {X -188.054,Y -220.761,Z 202.243,A 49.574,B 90.000,C 0.000} C_DIS
LIN {X -188.682,Y -220.225,Z 200.600,A 49.411,B 90.000,C 0.000} C_DIS
LIN {X -189.276,Y -219.715,Z 198.226,A 49.256,B 90.000,C 0.000} C_DIS
LIN {X -189.727,Y -219.325,Z 195.798,A 49.139,B 90.000,C 0.000} C_DIS
LIN {X -190.126,Y -218.980,Z 193.354,A 49.034,B 90.000,C 0.000} C_DIS
LIN {X -190.395,Y -218.746,Z 190.880,A 48.964,B 90.000,C 0.000} C_DIS
LIN {X -190.640,Y -218.533,Z 188.401,A 48.900,B 90.000,C 0.000} C_DIS
LIN {X -190.936,Y -218.274,Z 185.932,A 48.822,B 90.000,C 0.000} C_DIS
LIN {X -191.363,Y -217.900,Z 183.498,A 48.710,B 90.000,C 0.000} C_DIS
LIN {X -191.489,Y -217.789,Z 182.898,A 48.677,B 90.000,C 0.000} C_DIS
LIN {X -191.950,Y -217.383,Z 181.414,A 48.555,B 90.000,C 0.000} C_DIS
LIN {X -192.463,Y -216.928,Z 180.196,A 48.420,B 90.000,C 0.000} C_DIS
LIN {X -193.666,Y -215.855,Z 178.285,A 48.101,B 90.000,C 0.000} C_DIS
LIN {X -194.056,Y -215.505,Z 177.735,A 47.998,B 90.000,C 0.000} C_DIS
LIN {X -194.958,Y -214.689,Z 176.809,A 47.758,B 90.000,C 0.000} C_DIS
LIN {X -196.583,Y -213.201,Z 175.628,A 47.322,B 90.000,C 0.000} C_DIS
LIN {X -198.263,Y -211.637,Z 174.638,A 46.869,B 90.000,C 0.000} C_DIS
LIN {X -198.807,Y -211.130,Z 174.329,A 46.722,B 90.000,C 0.000} C_DIS
LIN {X -200.563,Y -209.461,Z 173.711,A 46.243,B 90.000,C 0.000} C_DIS
LIN {X -202.305,Y -207.777,Z 173.094,A 45.765,B 90.000,C 0.000} C_DIS
LIN {X -203.458,Y -206.652,Z 172.712,A 45.446,B 90.000,C 0.000} C_DIS
LIN {X -203.805,Y -206.310,Z 172.345,A 45.350,B 90.000,C 0.000} C_DIS
LIN {X -204.186,Y -205.933,Z 171.515,A 45.244,B 90.000,C 0.000} C_DIS
LIN {X -204.893,Y -205.229,Z 169.222,A 45.047,B 90.000,C 0.000} C_DIS
LIN {X -205.489,Y -204.631,Z 166.869,A 44.880,B 90.000,C 0.000} C_DIS
LIN {X -205.576,Y -204.544,Z 166.515,A 44.856,B 90.000,C 0.000} C_DIS
LIN {X -205.721,Y -204.399,Z 165.284,A 44.815,B 90.000,C 0.000} C_DIS
LIN {X -205.695,Y -204.425,Z 164.255,A 44.823,B 90.000,C 0.000} C_DIS
LIN {X -205.556,Y -204.564,Z 163.699,A 44.861,B 90.000,C 0.000} C_DIS
LIN {X -205.332,Y -204.789,Z 163.219,A 44.924,B 90.000,C 0.000} C_DIS
LIN {X -205.010,Y -205.112,Z 162.798,A 45.014,B 90.000,C 0.000} C_DIS
LIN {X -203.901,Y -206.214,Z 161.897,A 45.323,B 90.000,C 0.000} C_DIS
LIN {X -203.504,Y -206.606,Z 161.701,A 45.433,B 90.000,C 0.000} C_DIS
LIN {X -203.260,Y -206.846,Z 161.838,A 45.501,B 90.000,C 0.000} C_DIS
LIN {X -202.990,Y -207.111,Z 162.272,A 45.576,B 90.000,C 0.000} C_DIS
LIN {X -202.186,Y -207.895,Z 164.505,A 45.798,B 90.000,C 0.000} C_DIS
LIN {X -201.382,Y -208.674,Z 166.740,A 46.019,B 90.000,C 0.000} C_DIS
LIN {X -201.122,Y -208.925,Z 167.461,A 46.090,B 90.000,C 0.000} C_DIS
LIN {X -200.862,Y -209.175,Z 167.721,A 46.161,B 90.000,C 0.000} C_DIS
LIN {X -200.472,Y -209.550,Z 167.961,A 46.268,B 90.000,C 0.000} C_DIS
LIN {X -199.643,Y -210.339,Z 168.188,A 46.494,B 90.000,C 0.000} C_DIS
LIN {X -197.824,Y -212.049,Z 168.313,A 46.988,B 90.000,C 0.000} C_DIS
LIN {X -195.990,Y -213.747,Z 168.392,A 47.481,B 90.000,C 0.000} C_DIS
LIN {X -195.057,Y -214.599,Z 168.376,A 47.731,B 90.000,C 0.000} C_DIS
LIN {X -194.485,Y -215.118,Z 168.173,A 47.884,B 90.000,C 0.000} C_DIS
LIN {X -194.137,Y -215.432,Z 167.831,A 47.976,B 90.000,C 0.000} C_DIS
LIN {X -193.683,Y -215.840,Z 167.114,A 48.097,B 90.000,C 0.000} C_DIS
LIN {X -192.660,Y -216.752,Z 165.024,A 48.368,B 90.000,C 0.000} C_DIS
LIN {X -191.641,Y -217.654,Z 162.926,A 48.637,B 90.000,C 0.000} C_DIS
LIN {X -191.280,Y -217.973,Z 162.178,A 48.732,B 90.000,C 0.000} C_DIS
LIN {X -190.082,Y -219.017,Z 160.248,A 49.046,B 90.000,C 0.000} C_DIS
LIN {X -189.838,Y -219.230,Z 159.863,A 49.110,B 90.000,C 0.000} C_DIS
LIN {X -189.497,Y -219.524,Z 159.117,A 49.199,B 90.000,C 0.000} C_DIS
LIN {X -189.285,Y -219.707,Z 158.276,A 49.254,B 90.000,C 0.000} C_DIS
LIN {X -189.134,Y -219.837,Z 157.148,A 49.293,B 90.000,C 0.000} C_DIS
LIN {X -189.060,Y -219.900,Z 154.650,A 49.313,B 90.000,C 0.000} C_DIS
LIN {X -189.134,Y -219.837,Z 152.152,A 49.293,B 90.000,C 0.000} C_DIS
LIN {X -189.297,Y -219.696,Z 149.662,A 49.251,B 90.000,C 0.000} C_DIS
LIN {X -189.455,Y -219.560,Z 147.170,A 49.210,B 90.000,C 0.000} C_DIS
LIN {X -189.493,Y -219.527,Z 146.566,A 49.200,B 90.000,C 0.000} C_DIS
LIN {X -189.341,Y -219.659,Z 144.074,A 49.239,B 90.000,C 0.000} C_DIS
LIN {X -189.314,Y -219.682,Z 143.284,A 49.246,B 90.000,C 0.000} C_DIS
LIN {X -189.158,Y -219.816,Z 142.976,A 49.287,B 90.000,C 0.000} C_DIS
LIN {X -187.920,Y -220.875,Z 141.080,A 49.609,B 90.000,C 0.000} C_DIS
LIN {X -186.688,Y -221.918,Z 139.171,A 49.928,B 90.000,C 0.000} C_DIS
LIN {X -186.662,Y -221.940,Z 139.129,A 49.935,B 90.000,C 0.000} C_DIS
LIN {X -186.424,Y -222.140,Z 138.505,A 49.996,B 90.000,C 0.000} C_DIS
LIN {X -186.382,Y -222.175,Z 137.922,A 50.007,B 90.000,C 0.000} C_DIS
LIN {X -186.410,Y -222.151,Z 137.498,A 49.999,B 90.000,C 0.000} C_DIS
LIN {X -186.544,Y -222.039,Z 137.069,A 49.965,B 90.000,C 0.000} C_DIS
LIN {X -186.850,Y -221.782,Z 136.484,A 49.886,B 90.000,C 0.000} C_DIS
LIN {X -188.184,Y -220.650,Z 134.699,A 49.540,B 90.000,C 0.000} C_DIS
LIN {X -188.969,Y -219.979,Z 133.637,A 49.336,B 90.000,C 0.000} C_DIS
LIN {X -189.208,Y -219.773,Z 133.219,A 49.274,B 90.000,C 0.000} C_DIS
LIN {X -189.337,Y -219.662,Z 132.868,A 49.240,B 90.000,C 0.000} C_DIS
LIN {X -189.412,Y -219.597,Z 132.407,A 49.221,B 90.000,C 0.000} C_DIS
LIN {X -189.378,Y -219.627,Z 131.960,A 49.230,B 90.000,C 0.000} C_DIS
LIN {X -189.241,Y -219.745,Z 131.558,A 49.265,B 90.000,C 0.000} C_DIS
LIN {X -189.007,Y -219.946,Z 131.229,A 49.326,B 90.000,C 0.000} C_DIS
LIN {X -187.613,Y -221.136,Z 130.427,A 49.689,B 90.000,C 0.000} C_DIS
LIN {X -187.221,Y -221.469,Z 130.011,A 49.790,B 90.000,C 0.000} C_DIS
LIN {X -186.815,Y -221.811,Z 129.286,A 49.895,B 90.000,C 0.000} C_DIS
LIN {X -186.619,Y -221.976,Z 128.558,A 49.946,B 90.000,C 0.000} C_DIS
LIN {X -186.656,Y -221.945,Z 128.107,A 49.936,B 90.000,C 0.000} C_DIS
LIN {X -186.831,Y -221.797,Z 127.675,A 49.891,B 90.000,C 0.000} C_DIS
LIN {X -187.133,Y -221.543,Z 127.284,A 49.813,B 90.000,C 0.000} C_DIS
LIN {X -187.548,Y -221.191,Z 126.953,A 49.705,B 90.000,C 0.000} C_DIS
LIN {X -188.292,Y -220.558,Z 126.664,A 49.512,B 90.000,C 0.000} C_DIS
LIN {X -189.164,Y -219.811,Z 126.607,A 49.285,B 90.000,C 0.000} C_DIS
LIN {X -190.067,Y -219.031,Z 126.775,A 49.050,B 90.000,C 0.000} C_DIS
LIN {X -190.904,Y -218.301,Z 127.162,A 48.830,B 90.000,C 0.000} C_DIS
LIN {X -191.285,Y -217.968,Z 127.469,A 48.730,B 90.000,C 0.000} C_DIS
LIN {X -192.616,Y -216.793,Z 128.970,A 48.380,B 90.000,C 0.000} C_DIS
LIN {X -193.291,Y -216.191,Z 129.550,A 48.201,B 90.000,C 0.000} C_DIS
LIN {X -193.554,Y -215.956,Z 129.720,A 48.131,B 90.000,C 0.000} C_DIS
LIN {X -193.678,Y -215.845,Z 129.702,A 48.098,B 90.000,C 0.000} C_DIS
LIN {X -193.788,Y -215.745,Z 127.236,A 48.069,B 90.000,C 0.000} C_DIS
LIN {X -194.103,Y -215.462,Z 126.083,A 47.985,B 90.000,C 0.000} C_DIS
LIN {X -194.416,Y -215.180,Z 125.407,A 47.902,B 90.000,C 0.000} C_DIS
LIN {X -194.826,Y -214.809,Z 124.853,A 47.793,B 90.000,C 0.000} C_DIS
LIN {X -195.351,Y -214.332,Z 124.401,A 47.653,B 90.000,C 0.000} C_DIS
LIN {X -196.004,Y -213.735,Z 124.035,A 47.478,B 90.000,C 0.000} C_DIS
LIN {X -196.784,Y -213.016,Z 123.751,A 47.268,B 90.000,C 0.000} C_DIS
LIN {X -197.620,Y -212.241,Z 123.582,A 47.043,B 90.000,C 0.000} C_DIS
LIN {X -198.410,Y -211.503,Z 123.560,A 46.829,B 90.000,C 0.000} C_DIS
LIN {X -199.108,Y -210.846,Z 123.719,A 46.640,B 90.000,C 0.000} C_DIS
LIN {X -199.675,Y -210.309,Z 123.966,A 46.486,B 90.000,C 0.000} C_DIS
LIN {X -200.147,Y -209.860,Z 124.319,A 46.357,B 90.000,C 0.000} C_DIS
LIN {X -200.558,Y -209.467,Z 124.798,A 46.245,B 90.000,C 0.000} C_DIS
LIN {X -200.980,Y -209.062,Z 125.590,A 46.129,B 90.000,C 0.000} C_DIS
LIN {X -201.312,Y -208.742,Z 126.725,A 46.038,B 90.000,C 0.000} C_DIS
LIN {X -201.468,Y -208.592,Z 127.575,A 45.995,B 90.000,C 0.000} C_DIS
LIN {X -201.547,Y -208.516,Z 128.408,A 45.974,B 90.000,C 0.000} C_DIS
LIN {X -201.548,Y -208.515,Z 129.167,A 45.973,B 90.000,C 0.000} C_DIS
LIN {X -201.440,Y -208.619,Z 130.066,A 46.003,B 90.000,C 0.000} C_DIS
LIN {X -201.835,Y -208.237,Z 129.890,A 45.895,B 90.000,C 0.000} C_DIS
LIN {X -202.884,Y -207.215,Z 129.170,A 45.605,B 90.000,C 0.000} C_DIS
LIN {X -204.304,Y -205.814,Z 127.663,A 45.211,B 90.000,C 0.000} C_DIS
LIN {X -204.732,Y -205.390,Z 127.194,A 45.092,B 90.000,C 0.000} C_DIS
LIN {X -205.294,Y -204.827,Z 126.844,A 44.935,B 90.000,C 0.000} C_DIS
LIN {X -206.113,Y -204.004,Z 126.614,A 44.705,B 90.000,C 0.000} C_DIS
LIN {X -207.863,Y -202.220,Z 126.527,A 44.212,B 90.000,C 0.000} C_DIS
LIN {X -207.932,Y -202.149,Z 126.529,A 44.192,B 90.000,C 0.000} C_DIS
LIN {X -208.601,Y -201.459,Z 126.690,A 44.002,B 90.000,C 0.000} C_DIS
LIN {X -208.848,Y -201.203,Z 126.861,A 43.932,B 90.000,C 0.000} C_DIS
LIN {X -209.068,Y -200.974,Z 127.141,A 43.869,B 90.000,C 0.000} C_DIS
LIN {X -209.459,Y -200.566,Z 128.088,A 43.757,B 90.000,C 0.000} C_DIS
LIN {X -209.762,Y -200.250,Z 129.265,A 43.671,B 90.000,C 0.000} C_DIS
